LIN {X 0,Y 404.141,Z 498.144,A -85,B 0,C 180,E1 -10778.58,E2 -10778.58} C_VEL
LIN {X 0,Y 404.211,Z 498.134,A -85,B 0,C 180,E1 -10781.762,E2 -10781.762} C_VEL
LIN {X 0,Y 404.208,Z 498.138,A -85,B 0,C 180,E1 -10784.882,E2 -10784.882} C_VEL
LIN {X 0,Y 404.259,Z 498.127,A -85,B 0,C 180,E1 -10787.958,E2 -10787.958} C_VEL
LIN {X 0,Y 404.268,Z 498.129,A -85,B 0,C 180,E1 -10790.998,E2 -10790.998} C_VEL
LIN {X 0,Y 404.394,Z 498.111,A -85,B 0,C 180,E1 -10794.014,E2 -10794.014} C_VEL
LIN {X 0,Y 404.48,Z 498.1,A -85,B 0,C 180,E1 -10798.008,E2 -10798.008} C_VEL
LIN {X 0,Y 404.607,Z 498.084,A -85,B 0,C 180,E1 -10800,E2 -10800} C_VEL
LIN {X 0,Y 404.404,Z 498.112,A -85,B 0,C 180,E1 -10802.988,E2 -10802.988} C_VEL
LIN {X 0,Y 404.384,Z 498.112,A -85,B 0,C 180,E1 -10805.985,E2 -10805.985} C_VEL
LIN {X 0,Y 404.292,Z 498.126,A -85,B 0,C 180,E1 -10809.001,E2 -10809.001} C_VEL
LIN {X 0,Y 404.271,Z 498.126,A -85,B 0,C 180,E1 -10812.041,E2 -10812.041} C_VEL
LIN {X 0,Y 404.209,Z 498.136,A -85,B 0,C 180,E1 -10815.118,E2 -10815.118} C_VEL
LIN {X 0,Y 404.206,Z 498.135,A -85,B 0,C 180,E1 -10818.238,E2 -10818.238} C_VEL
LIN {X 0,Y 404.14,Z 498.144,A -85,B 0,C 180,E1 -10821.419,E2 -10821.419} C_VEL
LIN {X 0,Y 404.168,Z 498.142,A -85,B 0,C 180,E1 -10824.666,E2 -10824.666} C_VEL
LIN {X 0,Y 404.131,Z 498.144,A -85,B 0,C 180,E1 -10828.004,E2 -10828.004} C_VEL
LIN {X 0,Y 404.145,Z 498.143,A -85,B 0,C 180,E1 -10830.285,E2 -10830.285} C_VEL
LIN {X 0,Y 404.145,Z 498.142,A -85,B 0,C 180,E1 -10833.812,E2 -10833.812} C_VEL
LIN {X 0,Y 404.136,Z 498.147,A -85,B 0,C 180,E1 -10836.875,E2 -10836.875} C_VEL
LIN {X 0,Y 404.148,Z 498.145,A -85,B 0,C 180,E1 -10840.08,E2 -10840.08} C_VEL
LIN {X 0,Y 404.154,Z 498.142,A -85,B 0,C 180,E1 -10843.084,E2 -10843.084} C_VEL
LIN {X 0,Y 404.134,Z 498.16,A -85,B 0,C 180,E1 -10846.209,E2 -10846.209} C_VEL
LIN {X 0,Y 406.097,Z 507.927,A -85,B 0,C 180,E1 -10849.594,E2 -10849.594} C_VEL
LIN {X 0,Y 407.787,Z 516.569,A -85,B 0,C 180,E1 -10852.447,E2 -10852.447} C_VEL
LIN {X 0,Y 407.828,Z 520.057,A -85,B 0,C 180,E1 -10853.521,E2 -10853.521} C_VEL
LIN {X 0,Y 406.921,Z 529.958,A -85,B 0,C 180,E1 -10856.449,E2 -10856.449} C_VEL
LIN {X 0,Y 406.204,Z 539.849,A -85,B 0,C 180,E1 -10859.31,E2 -10859.31} C_VEL
LIN {X 0,Y 405.219,Z 553.615,A -85,B 0,C 180,E1 -10863.196,E2 -10863.196} C_VEL
LIN {X 0,Y 404.615,Z 565.406,A -85,B 0,C 180,E1 -10866.453,E2 -10866.453} C_VEL
LIN {X 0,Y 404,Z 579.554,A -85,B 0,C 180,E1 -10870.312,E2 -10870.312} C_VEL
LIN {X 0,Y 403.764,Z 586.685,A -85,B 0,C 180,E1 -10872.233,E2 -10872.233} C_VEL
LIN {X 0,Y 405.264,Z 601.573,A -85,B 0,C 180,E1 -10872.747,E2 -10872.747} C_VEL
LIN {X 0,Y 406.227,Z 614.758,A -85,B 0,C 180,E1 -10873.399,E2 -10873.399} C_VEL
LIN {X 0,Y 406.842,Z 625.399,A -85,B 0,C 180,E1 -10874.084,E2 -10874.084} C_VEL
LIN {X 0,Y 406.078,Z 636.59,A -85,B 0,C 180,E1 -10874.953,E2 -10874.953} C_VEL
LIN {X 0,Y 405.348,Z 646.907,A -85,B 0,C 180,E1 -10875.952,E2 -10875.952} C_VEL
LIN {X 0,Y 404.778,Z 654.204,A -85,B 0,C 180,E1 -10876.795,E2 -10876.795} C_VEL
LIN {X 0,Y 404.342,Z 660.999,A -85,B 0,C 180,E1 -10877.706,E2 -10877.706} C_VEL
LIN {X 0,Y 403.912,Z 668.935,A -85,B 0,C 180,E1 -10878.966,E2 -10878.966} C_VEL
LIN {X 0,Y 403.564,Z 676.692,A -85,B 0,C 180,E1 -10880.477,E2 -10880.477} C_VEL
LIN {X 0,Y 403.396,Z 682.935,A -85,B 0,C 180,E1 -10881.988,E2 -10881.988} C_VEL
LIN {X 0,Y 403.358,Z 687.287,A -85,B 0,C 180,E1 -10883.292,E2 -10883.292} C_VEL
LIN {X 0,Y 403.51,Z 691.675,A -85,B 0,C 180,E1 -10885.004,E2 -10885.004} C_VEL
LIN {X 0,Y 403.575,Z 693.612,A -85,B 0,C 180,E1 -10886.006,E2 -10886.006} C_VEL
LIN {X 0,Y 403.543,Z 695.082,A -85,B 0,C 180,E1 -10887.005,E2 -10887.005} C_VEL
LIN {X 0,Y 403.577,Z 696.088,A -85,B 0,C 180,E1 -10888.004,E2 -10888.004} C_VEL
LIN {X 0,Y 403.818,Z 696.903,A -85,B 0,C 180,E1 -10890,E2 -10890} C_VEL
LIN {X 0,Y 403.62,Z 696.63,A -85,B 0,C 180,E1 -10890.998,E2 -10890.998} C_VEL
LIN {X 0,Y 403.595,Z 695.93,A -85,B 0,C 180,E1 -10891.996,E2 -10891.996} C_VEL
LIN {X 0,Y 403.565,Z 694.822,A -85,B 0,C 180,E1 -10892.995,E2 -10892.995} C_VEL
LIN {X 0,Y 403.576,Z 692.346,A -85,B 0,C 180,E1 -10894.495,E2 -10894.495} C_VEL
LIN {X 0,Y 403.425,Z 688.813,A -85,B 0,C 180,E1 -10896,E2 -10896} C_VEL
LIN {X 0,Y 403.407,Z 684.179,A -85,B 0,C 180,E1 -10897.508,E2 -10897.508} C_VEL
LIN {X 0,Y 403.496,Z 678.319,A -85,B 0,C 180,E1 -10899.019,E2 -10899.019} C_VEL
LIN {X 0,Y 403.739,Z 671.062,A -85,B 0,C 180,E1 -10900.532,E2 -10900.532} C_VEL
LIN {X 0,Y 404.148,Z 663.731,A -85,B 0,C 180,E1 -10901.79,E2 -10901.79} C_VEL
LIN {X 0,Y 404.728,Z 654.992,A -85,B 0,C 180,E1 -10903.047,E2 -10903.047} C_VEL
LIN {X 0,Y 405.372,Z 645.507,A -85,B 0,C 180,E1 -10904.175,E2 -10904.175} C_VEL
LIN {X 0,Y 406.273,Z 633.869,A -85,B 0,C 180,E1 -10905.296,E2 -10905.296} C_VEL
LIN {X 0,Y 406.924,Z 624.366,A -85,B 0,C 180,E1 -10906.042,E2 -10906.042} C_VEL
LIN {X 0,Y 406.386,Z 614.636,A -85,B 0,C 180,E1 -10906.709,E2 -10906.709} C_VEL
LIN {X 0,Y 405.749,Z 600.808,A -85,B 0,C 180,E1 -10907.444,E2 -10907.444} C_VEL
LIN {X 0,Y 404.415,Z 587.584,A -85,B 0,C 180,E1 -10907.975,E2 -10907.975} C_VEL
LIN {X 0,Y 403.758,Z 582.357,A -85,B 0,C 180,E1 -10908.164,E2 -10908.164} C_VEL
LIN {X 0,Y 404.09,Z 568.944,A -85,B 0,C 180,E1 -10911.69,E2 -10911.69} C_VEL
LIN {X 0,Y 404.645,Z 555.051,A -85,B 0,C 180,E1 -10915.424,E2 -10915.424} C_VEL
LIN {X 0,Y 405.304,Z 541.989,A -85,B 0,C 180,E1 -10919.047,E2 -10919.047} C_VEL
LIN {X 0,Y 406.089,Z 530.165,A -85,B 0,C 180,E1 -10922.446,E2 -10922.446} C_VEL
LIN {X 0,Y 407.046,Z 518.566,A -85,B 0,C 180,E1 -10925.948,E2 -10925.948} C_VEL
LIN {X 0,Y 407.158,Z 513.919,A -85,B 0,C 180,E1 -10927.438,E2 -10927.438} C_VEL
LIN {X 0,Y 405.718,Z 505.699,A -85,B 0,C 180,E1 -10930.343,E2 -10930.343} C_VEL
LIN {X 0,Y 404.151,Z 498.147,A -85,B 0,C 180,E1 -10933.287,E2 -10933.287} C_VEL
LIN {X 0,Y 404.156,Z 498.146,A -85,B 0,C 180,E1 -10936.916,E2 -10936.916} C_VEL
LIN {X 0,Y 404.171,Z 498.141,A -85,B 0,C 180,E1 -10939.956,E2 -10939.956} C_VEL
LIN {X 0,Y 404.138,Z 498.145,A -85,B 0,C 180,E1 -10943.125,E2 -10943.125} C_VEL
LIN {X 0,Y 404.147,Z 498.142,A -85,B 0,C 180,E1 -10946.188,E2 -10946.188} C_VEL
LIN {X 0,Y 404.148,Z 498.144,A -85,B 0,C 180,E1 -10949.715,E2 -10949.715} C_VEL
LIN {X 0,Y 404.198,Z 498.133,A -85,B 0,C 180,E1 -10953.123,E2 -10953.123} C_VEL
LIN {X 0,Y 404.18,Z 498.137,A -85,B 0,C 180,E1 -10955.335,E2 -10955.335} C_VEL
LIN {X 0,Y 404.142,Z 498.14,A -85,B 0,C 180,E1 -10958.581,E2 -10958.581} C_VEL
LIN {X 0,Y 404.212,Z 498.132,A -85,B 0,C 180,E1 -10961.762,E2 -10961.762} C_VEL
LIN {X 0,Y 404.21,Z 498.132,A -85,B 0,C 180,E1 -10964.882,E2 -10964.882} C_VEL
LIN {X 0,Y 404.26,Z 498.128,A -85,B 0,C 180,E1 -10967.959,E2 -10967.959} C_VEL
LIN {X 0,Y 404.437,Z 498.103,A -85,B 0,C 180,E1 -10972.1,E2 -10972.1} C_VEL
LIN {X 0,Y 404.428,Z 498.108,A -85,B 0,C 180,E1 -10974.015,E2 -10974.015} C_VEL
LIN {X 0,Y 404.482,Z 498.101,A -85,B 0,C 180,E1 -10978.009,E2 -10978.009} C_VEL
LIN {X 0,Y 404.612,Z 498.086,A -85,B 0,C 180,E1 -10980,E2 -10980} C_VEL
LIN {X 0,Y 404.419,Z 498.111,A -85,B 0,C 180,E1 -10982.989,E2 -10982.989} C_VEL
LIN {X 0,Y 404.35,Z 498.114,A -85,B 0,C 180,E1 -10986.534,E2 -10986.534} C_VEL
LIN {X 0,Y 404.293,Z 498.123,A -85,B 0,C 180,E1 -10989.001,E2 -10989.001} C_VEL
LIN {X 0,Y 404.261,Z 498.131,A -85,B 0,C 180,E1 -10992.042,E2 -10992.042} C_VEL
LIN {X 0,Y 404.213,Z 498.136,A -85,B 0,C 180,E1 -10995.118,E2 -10995.118} C_VEL
LIN {X 0,Y 404.259,Z 498.134,A -85,B 0,C 180,E1 -10996.745,E2 -10996.745} C_VEL
LIN {X 0,Y 408.406,Z 510.86,A -85,B 0,C 180,E1 -10997.786,E2 -10997.786} C_VEL
LIN {X 0,Y 409.398,Z 514.616,A -85,B 0,C 180,E1 -10998.129,E2 -10998.129} C_VEL
LIN {X 0,Y 408.929,Z 525.453,A -85,B 0,C 180,E1 -10999.059,E2 -10999.059} C_VEL
LIN {X 0,Y 408.19,Z 535.615,A -85,B 0,C 180,E1 -11000.142,E2 -11000.142} C_VEL
LIN {X 0,Y 407.382,Z 545.671,A -85,B 0,C 180,E1 -11001.479,E2 -11001.479} C_VEL
LIN {X 0,Y 406.617,Z 554.21,A -85,B 0,C 180,E1 -11002.886,E2 -11002.886} C_VEL
LIN {X 0,Y 406.019,Z 560.977,A -85,B 0,C 180,E1 -11004.274,E2 -11004.274} C_VEL
LIN {X 0,Y 405.502,Z 566.524,A -85,B 0,C 180,E1 -11005.677,E2 -11005.677} C_VEL
LIN {X 0,Y 405.001,Z 571.46,A -85,B 0,C 180,E1 -11007.261,E2 -11007.261} C_VEL
LIN {X 0,Y 404.571,Z 575.675,A -85,B 0,C 180,E1 -11009.105,E2 -11009.105} C_VEL
LIN {X 0,Y 404.343,Z 577.544,A -85,B 0,C 180,E1 -11010.269,E2 -11010.269} C_VEL
LIN {X 0,Y 404.164,Z 578.987,A -85,B 0,C 180,E1 -11011.563,E2 -11011.563} C_VEL
LIN {X 0,Y 404.021,Z 579.832,A -85,B 0,C 180,E1 -11013.387,E2 -11013.387} C_VEL
LIN {X 0,Y 403.999,Z 579.409,A -85,B 0,C 180,E1 -11015.153,E2 -11015.153} C_VEL
LIN {X 0,Y 404.036,Z 577.843,A -85,B 0,C 180,E1 -11016.855,E2 -11016.855} C_VEL
LIN {X 0,Y 404.242,Z 574.712,A -85,B 0,C 180,E1 -11018.748,E2 -11018.748} C_VEL
LIN {X 0,Y 404.633,Z 569.886,A -85,B 0,C 180,E1 -11020.661,E2 -11020.661} C_VEL
LIN {X 0,Y 404.958,Z 565.075,A -85,B 0,C 180,E1 -11022.102,E2 -11022.102} C_VEL
LIN {X 0,Y 405.363,Z 559.33,A -85,B 0,C 180,E1 -11023.489,E2 -11023.489} C_VEL
LIN {X 0,Y 405.978,Z 551.93,A -85,B 0,C 180,E1 -11024.94,E2 -11024.94} C_VEL
LIN {X 0,Y 406.592,Z 543.052,A -85,B 0,C 180,E1 -11026.347,E2 -11026.347} C_VEL
LIN {X 0,Y 407.271,Z 533.218,A -85,B 0,C 180,E1 -11027.609,E2 -11027.609} C_VEL
LIN {X 0,Y 407.904,Z 522.41,A -85,B 0,C 180,E1 -11028.733,E2 -11028.733} C_VEL
LIN {X 0,Y 408.384,Z 513.674,A -85,B 0,C 180,E1 -11029.47,E2 -11029.47} C_VEL
LIN {X 0,Y 405.738,Z 503.665,A -85,B 0,C 180,E1 -11030.302,E2 -11030.302} C_VEL
LIN {X 0,Y 404.159,Z 498.143,A -85,B 0,C 180,E1 -11030.722,E2 -11030.722} C_VEL
LIN {X 0,Y 404.146,Z 498.145,A -85,B 0,C 180,E1 -11033.754,E2 -11033.754} C_VEL
LIN {X 0,Y 404.176,Z 498.137,A -85,B 0,C 180,E1 -11036.58,E2 -11036.58} C_VEL
LIN {X 0,Y 404.168,Z 498.138,A -85,B 0,C 180,E1 -11040.395,E2 -11040.395} C_VEL
LIN {X 0,Y 404.199,Z 498.138,A -85,B 0,C 180,E1 -11043.123,E2 -11043.123} C_VEL
LIN {X 0,Y 404.175,Z 498.141,A -85,B 0,C 180,E1 -11045.334,E2 -11045.334} C_VEL
LIN {X 0,Y 404.144,Z 498.142,A -85,B 0,C 180,E1 -11048.581,E2 -11048.581} C_VEL
LIN {X 0,Y 404.21,Z 498.136,A -85,B 0,C 180,E1 -11051.762,E2 -11051.762} C_VEL
LIN {X 0,Y 404.211,Z 498.135,A -85,B 0,C 180,E1 -11054.882,E2 -11054.882} C_VEL
LIN {X 0,Y 404.262,Z 498.128,A -85,B 0,C 180,E1 -11057.958,E2 -11057.958} C_VEL
LIN {X 0,Y 404.272,Z 498.129,A -85,B 0,C 180,E1 -11060.998,E2 -11060.998} C_VEL
LIN {X 0,Y 404.387,Z 498.112,A -85,B 0,C 180,E1 -11064.014,E2 -11064.014} C_VEL
LIN {X 0,Y 404.485,Z 498.1,A -85,B 0,C 180,E1 -11068.008,E2 -11068.008} C_VEL
LIN {X 0,Y 404.606,Z 498.085,A -85,B 0,C 180,E1 -11070,E2 -11070} C_VEL
LIN {X 0,Y 404.413,Z 498.111,A -85,B 0,C 180,E1 -11072.988,E2 -11072.988} C_VEL
LIN {X 0,Y 404.386,Z 498.112,A -85,B 0,C 180,E1 -11075.985,E2 -11075.985} C_VEL
LIN {X 0,Y 404.271,Z 498.129,A -85,B 0,C 180,E1 -11079.001,E2 -11079.001} C_VEL
LIN {X 0,Y 404.261,Z 498.127,A -85,B 0,C 180,E1 -11082.041,E2 -11082.041} C_VEL
LIN {X 0,Y 404.205,Z 498.136,A -85,B 0,C 180,E1 -11085.267,E2 -11085.267} C_VEL
LIN {X 0,Y 403.533,Z 498.219,A -85,B 0,C 180,E1 -11086.098,E2 -11086.098} C_VEL
LIN {X 0,Y 400.696,Z 498.575,A -85,B 0,C 180,E1 -11087.449,E2 -11087.449} C_VEL
LIN {X 0,Y 398.29,Z 498.876,A -85,B 0,C 180,E1 -11088.54,E2 -11088.54} C_VEL
LIN {X 0,Y 397.243,Z 499.004,A -85,B 0,C 180,E1 -11089.384,E2 -11089.384} C_VEL
LIN {X 0,Y 397.15,Z 499.014,A -85,B 0,C 180,E1 -11089.67,E2 -11089.67} C_VEL
LIN {X 0,Y 397.139,Z 499.017,A -85,B 0,C 180,E1 -11093.04,E2 -11093.04} C_VEL
LIN {X 0,Y 397.107,Z 499.017,A -85,B 0,C 180,E1 -11096.26,E2 -11096.26} C_VEL
LIN {X 0,Y 397.123,Z 499.018,A -85,B 0,C 180,E1 -11099.704,E2 -11099.704} C_VEL
LIN {X 0,Y 397.118,Z 499.02,A -85,B 0,C 180,E1 -11103.273,E2 -11103.273} C_VEL
LIN {X 0,Y 397.111,Z 499.019,A -85,B 0,C 180,E1 -11105.734,E2 -11105.734} C_VEL
LIN {X 0,Y 397.098,Z 499.022,A -85,B 0,C 180,E1 -11108.855,E2 -11108.855} C_VEL
LIN {X 0,Y 397.06,Z 499.024,A -85,B 0,C 180,E1 -11112.268,E2 -11112.268} C_VEL
LIN {X 0,Y 397.09,Z 499.024,A -85,B 0,C 180,E1 -11115.069,E2 -11115.069} C_VEL
LIN {X 0,Y 397.065,Z 499.023,A -85,B 0,C 180,E1 -11118.022,E2 -11118.022} C_VEL
LIN {X 0,Y 397.127,Z 499.019,A -85,B 0,C 180,E1 -11121.139,E2 -11121.139} C_VEL
LIN {X 0,Y 397.122,Z 499.018,A -85,B 0,C 180,E1 -11124.496,E2 -11124.496} C_VEL
LIN {X 0,Y 397.081,Z 499.022,A -85,B 0,C 180,E1 -11127.928,E2 -11127.928} C_VEL
LIN {X 0,Y 397.125,Z 499.017,A -85,B 0,C 180,E1 -11131.456,E2 -11131.456} C_VEL
LIN {X 0,Y 397.154,Z 499.014,A -85,B 0,C 180,E1 -11134.488,E2 -11134.488} C_VEL
LIN {X 0,Y 397.099,Z 499.018,A -85,B 0,C 180,E1 -11138.181,E2 -11138.181} C_VEL
LIN {X 0,Y 397.164,Z 499.013,A -85,B 0,C 180,E1 -11141.426,E2 -11141.426} C_VEL
LIN {X 0,Y 397.181,Z 499.011,A -85,B 0,C 180,E1 -11144.608,E2 -11144.608} C_VEL
LIN {X 0,Y 397.222,Z 499.004,A -85,B 0,C 180,E1 -11147.742,E2 -11147.742} C_VEL
LIN {X 0,Y 397.238,Z 499.006,A -85,B 0,C 180,E1 -11150.837,E2 -11150.837} C_VEL
LIN {X 0,Y 397.346,Z 498.988,A -85,B 0,C 180,E1 -11153.908,E2 -11153.908} C_VEL
LIN {X 0,Y 397.449,Z 498.976,A -85,B 0,C 180,E1 -11157.973,E2 -11157.973} C_VEL
LIN {X 0,Y 397.577,Z 498.96,A -85,B 0,C 180,E1 -11160,E2 -11160} C_VEL
LIN {X 0,Y 397.337,Z 498.992,A -85,B 0,C 180,E1 -11163.041,E2 -11163.041} C_VEL
LIN {X 0,Y 397.335,Z 498.99,A -85,B 0,C 180,E1 -11166.092,E2 -11166.092} C_VEL
LIN {X 0,Y 397.254,Z 499.002,A -85,B 0,C 180,E1 -11169.162,E2 -11169.162} C_VEL
LIN {X 0,Y 397.23,Z 499.004,A -85,B 0,C 180,E1 -11172.258,E2 -11172.258} C_VEL
LIN {X 0,Y 397.181,Z 499.011,A -85,B 0,C 180,E1 -11175.392,E2 -11175.392} C_VEL
LIN {X 0,Y 397.16,Z 499.014,A -85,B 0,C 180,E1 -11178.573,E2 -11178.573} C_VEL
LIN {X 0,Y 397.098,Z 499.019,A -85,B 0,C 180,E1 -11181.818,E2 -11181.818} C_VEL
LIN {X 0,Y 397.125,Z 499.018,A -85,B 0,C 180,E1 -11185.134,E2 -11185.134} C_VEL
LIN {X 0,Y 397.079,Z 499.025,A -85,B 0,C 180,E1 -11188.547,E2 -11188.547} C_VEL
LIN {X 0,Y 397.082,Z 499.02,A -85,B 0,C 180,E1 -11191.836,E2 -11191.836} C_VEL
LIN {X 0,Y 397.126,Z 499.019,A -85,B 0,C 180,E1 -11194.493,E2 -11194.493} C_VEL
LIN {X 0,Y 397.099,Z 499.02,A -85,B 0,C 180,E1 -11198.275,E2 -11198.275} C_VEL
LIN {X 0,Y 397.09,Z 499.024,A -85,B 0,C 180,E1 -11200.909,E2 -11200.909} C_VEL
LIN {X 0,Y 397.102,Z 499.019,A -85,B 0,C 180,E1 -11203.648,E2 -11203.648} C_VEL
LIN {X 0,Y 397.122,Z 499.123,A -85,B 0,C 180,E1 -11205.91,E2 -11205.91} C_VEL
LIN {X 0,Y 399.047,Z 508.804,A -85,B 0,C 180,E1 -11209.334,E2 -11209.334} C_VEL
LIN {X 0,Y 400.847,Z 518.125,A -85,B 0,C 180,E1 -11212.463,E2 -11212.463} C_VEL
LIN {X 0,Y 400.738,Z 522.352,A -85,B 0,C 180,E1 -11213.778,E2 -11213.778} C_VEL
LIN {X 0,Y 399.751,Z 532.996,A -85,B 0,C 180,E1 -11216.975,E2 -11216.975} C_VEL
LIN {X 0,Y 398.957,Z 543.459,A -85,B 0,C 180,E1 -11220.044,E2 -11220.044} C_VEL
LIN {X 0,Y 398.034,Z 556.584,A -85,B 0,C 180,E1 -11223.806,E2 -11223.806} C_VEL
LIN {X 0,Y 397.407,Z 568.298,A -85,B 0,C 180,E1 -11227.104,E2 -11227.104} C_VEL
LIN {X 0,Y 396.82,Z 581.904,A -85,B 0,C 180,E1 -11230.874,E2 -11230.874} C_VEL
LIN {X 0,Y 396.676,Z 585.78,A -85,B 0,C 180,E1 -11231.938,E2 -11231.938} C_VEL
LIN {X 0,Y 398.191,Z 600.26,A -85,B 0,C 180,E1 -11232.449,E2 -11232.449} C_VEL
LIN {X 0,Y 399.15,Z 613.084,A -85,B 0,C 180,E1 -11233.087,E2 -11233.087} C_VEL
LIN {X 0,Y 399.754,Z 623.972,A -85,B 0,C 180,E1 -11233.794,E2 -11233.794} C_VEL
LIN {X 0,Y 399.239,Z 633.846,A -85,B 0,C 180,E1 -11234.559,E2 -11234.559} C_VEL
LIN {X 0,Y 398.35,Z 645.631,A -85,B 0,C 180,E1 -11235.7,E2 -11235.7} C_VEL
LIN {X 0,Y 397.71,Z 654.208,A -85,B 0,C 180,E1 -11236.719,E2 -11236.719} C_VEL
LIN {X 0,Y 397.111,Z 663.135,A -85,B 0,C 180,E1 -11237.998,E2 -11237.998} C_VEL
LIN {X 0,Y 396.72,Z 670.534,A -85,B 0,C 180,E1 -11239.28,E2 -11239.28} C_VEL
LIN {X 0,Y 396.406,Z 677.823,A -85,B 0,C 180,E1 -11240.819,E2 -11240.819} C_VEL
LIN {X 0,Y 396.309,Z 683.639,A -85,B 0,C 180,E1 -11242.357,E2 -11242.357} C_VEL
LIN {X 0,Y 396.331,Z 688.204,A -85,B 0,C 180,E1 -11243.893,E2 -11243.893} C_VEL
LIN {X 0,Y 396.464,Z 690.607,A -85,B 0,C 180,E1 -11244.915,E2 -11244.915} C_VEL
LIN {X 0,Y 396.539,Z 692.553,A -85,B 0,C 180,E1 -11245.935,E2 -11245.935} C_VEL
LIN {X 0,Y 396.506,Z 694.036,A -85,B 0,C 180,E1 -11246.952,E2 -11246.952} C_VEL
LIN {X 0,Y 396.542,Z 695.051,A -85,B 0,C 180,E1 -11247.969,E2 -11247.969} C_VEL
LIN {X 0,Y 396.795,Z 695.873,A -85,B 0,C 180,E1 -11250,E2 -11250} C_VEL
LIN {X 0,Y 396.589,Z 695.609,A -85,B 0,C 180,E1 -11251.016,E2 -11251.016} C_VEL
LIN {X 0,Y 396.556,Z 694.912,A -85,B 0,C 180,E1 -11252.031,E2 -11252.031} C_VEL
LIN {X 0,Y 396.572,Z 692.289,A -85,B 0,C 180,E1 -11254.065,E2 -11254.065} C_VEL
LIN {X 0,Y 396.373,Z 689.098,A -85,B 0,C 180,E1 -11255.596,E2 -11255.596} C_VEL
LIN {X 0,Y 396.34,Z 684.847,A -85,B 0,C 180,E1 -11257.13,E2 -11257.13} C_VEL
LIN {X 0,Y 396.411,Z 678.397,A -85,B 0,C 180,E1 -11258.924,E2 -11258.924} C_VEL
LIN {X 0,Y 396.625,Z 671.39,A -85,B 0,C 180,E1 -11260.465,E2 -11260.465} C_VEL
LIN {X 0,Y 397.113,Z 662.782,A -85,B 0,C 180,E1 -11262.002,E2 -11262.002} C_VEL
LIN {X 0,Y 397.662,Z 654.059,A -85,B 0,C 180,E1 -11263.283,E2 -11263.283} C_VEL
LIN {X 0,Y 398.556,Z 643.445,A -85,B 0,C 180,E1 -11264.553,E2 -11264.553} C_VEL
LIN {X 0,Y 399.413,Z 633.058,A -85,B 0,C 180,E1 -11265.565,E2 -11265.565} C_VEL
LIN {X 0,Y 399.956,Z 625.373,A -85,B 0,C 180,E1 -11266.198,E2 -11266.198} C_VEL
LIN {X 0,Y 399.455,Z 614.004,A -85,B 0,C 180,E1 -11267.008,E2 -11267.008} C_VEL
LIN {X 0,Y 398.847,Z 600.684,A -85,B 0,C 180,E1 -11267.747,E2 -11267.747} C_VEL
LIN {X 0,Y 397.502,Z 586.889,A -85,B 0,C 180,E1 -11268.332,E2 -11268.332} C_VEL
LIN {X 0,Y 396.685,Z 581.208,A -85,B 0,C 180,E1 -11268.53,E2 -11268.53} C_VEL
LIN {X 0,Y 397.056,Z 567.967,A -85,B 0,C 180,E1 -11272.095,E2 -11272.095} C_VEL
LIN {X 0,Y 397.642,Z 555.002,A -85,B 0,C 180,E1 -11275.659,E2 -11275.659} C_VEL
LIN {X 0,Y 398.254,Z 543.102,A -85,B 0,C 180,E1 -11279.032,E2 -11279.032} C_VEL
LIN {X 0,Y 399.132,Z 530.894,A -85,B 0,C 180,E1 -11282.624,E2 -11282.624} C_VEL
LIN {X 0,Y 400.103,Z 519.649,A -85,B 0,C 180,E1 -11286.098,E2 -11286.098} C_VEL
LIN {X 0,Y 400.33,Z 516.239,A -85,B 0,C 180,E1 -11287.199,E2 -11287.199} C_VEL
LIN {X 0,Y 399.018,Z 508.383,A -85,B 0,C 180,E1 -11290.008,E2 -11290.008} C_VEL
LIN {X 0,Y 397.547,Z 501.176,A -85,B 0,C 180,E1 -11292.829,E2 -11292.829} C_VEL
LIN {X 0,Y 397.106,Z 499.027,A -85,B 0,C 180,E1 -11293.736,E2 -11293.736} C_VEL
LIN {X 0,Y 397.105,Z 499.026,A -85,B 0,C 180,E1 -11296.521,E2 -11296.521} C_VEL
LIN {X 0,Y 397.116,Z 499.021,A -85,B 0,C 180,E1 -11300.423,E2 -11300.423} C_VEL
LIN {X 0,Y 397.11,Z 499.02,A -85,B 0,C 180,E1 -11304.266,E2 -11304.266} C_VEL
LIN {X 0,Y 397.117,Z 499.019,A -85,B 0,C 180,E1 -11306.727,E2 -11306.727} C_VEL
LIN {X 0,Y 397.127,Z 499.014,A -85,B 0,C 180,E1 -11310.296,E2 -11310.296} C_VEL
LIN {X 0,Y 397.197,Z 499.006,A -85,B 0,C 180,E1 -11312.61,E2 -11312.61} C_VEL
LIN {X 0,Y 397.135,Z 499.012,A -85,B 0,C 180,E1 -11315.982,E2 -11315.982} C_VEL
LIN {X 0,Y 397.142,Z 499.013,A -85,B 0,C 180,E1 -11319.705,E2 -11319.705} C_VEL
LIN {X 0,Y 397.185,Z 499.01,A -85,B 0,C 180,E1 -11322.845,E2 -11322.845} C_VEL
LIN {X 0,Y 397.232,Z 499.005,A -85,B 0,C 180,E1 -11326.703,E2 -11326.703} C_VEL
LIN {X 0,Y 397.221,Z 499.007,A -85,B 0,C 180,E1 -11329.809,E2 -11329.809} C_VEL
LIN {X 0,Y 397.369,Z 498.987,A -85,B 0,C 180,E1 -11332.889,E2 -11332.889} C_VEL
LIN {X 0,Y 397.253,Z 498.998,A -85,B 0,C 180,E1 -11334.925,E2 -11334.925} C_VEL
LIN {X 0,Y 397.45,Z 498.976,A -85,B 0,C 180,E1 -11337.974,E2 -11337.974} C_VEL
LIN {X 0,Y 397.581,Z 498.961,A -85,B 0,C 180,E1 -11340,E2 -11340} C_VEL
LIN {X 0,Y 397.378,Z 498.988,A -85,B 0,C 180,E1 -11343.042,E2 -11343.042} C_VEL
LIN {X 0,Y 397.306,Z 498.991,A -85,B 0,C 180,E1 -11346.527,E2 -11346.527} C_VEL
LIN {X 0,Y 397.256,Z 499,A -85,B 0,C 180,E1 -11349.162,E2 -11349.162} C_VEL
LIN {X 0,Y 397.224,Z 499.009,A -85,B 0,C 180,E1 -11352.258,E2 -11352.258} C_VEL
LIN {X 0,Y 397.191,Z 499.013,A -85,B 0,C 180,E1 -11355.918,E2 -11355.918} C_VEL
LIN {X 0,Y 397.217,Z 499.129,A -85,B 0,C 180,E1 -11356.379,E2 -11356.379} C_VEL
LIN {X 0,Y 401.529,Z 512.126,A -85,B 0,C 180,E1 -11357.469,E2 -11357.469} C_VEL
LIN {X 0,Y 402.748,Z 516.55,A -85,B 0,C 180,E1 -11357.887,E2 -11357.887} C_VEL
LIN {X 0,Y 402.127,Z 527.968,A -85,B 0,C 180,E1 -11358.907,E2 -11358.907} C_VEL
LIN {X 0,Y 401.341,Z 538.575,A -85,B 0,C 180,E1 -11360.1,E2 -11360.1} C_VEL
LIN {X 0,Y 400.526,Z 547.771,A -85,B 0,C 180,E1 -11361.378,E2 -11361.378} C_VEL
LIN {X 0,Y 399.735,Z 555.793,A -85,B 0,C 180,E1 -11362.756,E2 -11362.756} C_VEL
LIN {X 0,Y 398.97,Z 563.649,A -85,B 0,C 180,E1 -11364.454,E2 -11364.454} C_VEL
LIN {X 0,Y 398.343,Z 569.823,A -85,B 0,C 180,E1 -11366.173,E2 -11366.173} C_VEL
LIN {X 0,Y 397.843,Z 574.613,A -85,B 0,C 180,E1 -11367.961,E2 -11367.961} C_VEL
LIN {X 0,Y 397.436,Z 577.893,A -85,B 0,C 180,E1 -11369.679,E2 -11369.679} C_VEL
LIN {X 0,Y 397.259,Z 579.438,A -85,B 0,C 180,E1 -11370.867,E2 -11370.867} C_VEL
LIN {X 0,Y 397.087,Z 580.431,A -85,B 0,C 180,E1 -11372.071,E2 -11372.071} C_VEL
LIN {X 0,Y 397.006,Z 580.885,A -85,B 0,C 180,E1 -11373.693,E2 -11373.693} C_VEL
LIN {X 0,Y 397.002,Z 580.025,A -85,B 0,C 180,E1 -11375.746,E2 -11375.746} C_VEL
LIN {X 0,Y 397.043,Z 578.454,A -85,B 0,C 180,E1 -11377.199,E2 -11377.199} C_VEL
LIN {X 0,Y 397.238,Z 575.543,A -85,B 0,C 180,E1 -11378.88,E2 -11378.88} C_VEL
LIN {X 0,Y 397.663,Z 570.612,A -85,B 0,C 180,E1 -11380.838,E2 -11380.838} C_VEL
LIN {X 0,Y 398.085,Z 565.076,A -85,B 0,C 180,E1 -11382.477,E2 -11382.477} C_VEL
LIN {X 0,Y 398.64,Z 557.594,A -85,B 0,C 180,E1 -11384.195,E2 -11384.195} C_VEL
LIN {X 0,Y 399.292,Z 549.75,A -85,B 0,C 180,E1 -11385.635,E2 -11385.635} C_VEL
LIN {X 0,Y 399.971,Z 540.08,A -85,B 0,C 180,E1 -11387.072,E2 -11387.072} C_VEL
LIN {X 0,Y 400.688,Z 529.022,A -85,B 0,C 180,E1 -11388.385,E2 -11388.385} C_VEL
LIN {X 0,Y 401.335,Z 518.926,A -85,B 0,C 180,E1 -11389.348,E2 -11389.348} C_VEL
LIN {X 0,Y 401.318,Z 513.838,A -85,B 0,C 180,E1 -11389.776,E2 -11389.776} C_VEL
LIN {X 0,Y 398.034,Z 502.298,A -85,B 0,C 180,E1 -11390.734,E2 -11390.734} C_VEL
LIN {X 0,Y 397.112,Z 499.022,A -85,B 0,C 180,E1 -11390.978,E2 -11390.978} C_VEL
LIN {X 0,Y 397.124,Z 499.016,A -85,B 0,C 180,E1 -11394.497,E2 -11394.497} C_VEL
LIN {X 0,Y 397.084,Z 499.023,A -85,B 0,C 180,E1 -11397.929,E2 -11397.929} C_VEL
LIN {X 0,Y 397.127,Z 499.02,A -85,B 0,C 180,E1 -11401.456,E2 -11401.456} C_VEL
LIN {X 0,Y 397.156,Z 499.012,A -85,B 0,C 180,E1 -11404.488,E2 -11404.488} C_VEL
LIN {X 0,Y 397.101,Z 499.019,A -85,B 0,C 180,E1 -11408.181,E2 -11408.181} C_VEL
LIN {X 0,Y 397.163,Z 499.015,A -85,B 0,C 180,E1 -11411.426,E2 -11411.426} C_VEL
LIN {X 0,Y 397.184,Z 499.009,A -85,B 0,C 180,E1 -11414.608,E2 -11414.608} C_VEL
LIN {X 0,Y 397.225,Z 499.006,A -85,B 0,C 180,E1 -11417.742,E2 -11417.742} C_VEL
LIN {X 0,Y 397.241,Z 499.003,A -85,B 0,C 180,E1 -11420.838,E2 -11420.838} C_VEL
LIN {X 0,Y 397.338,Z 498.99,A -85,B 0,C 180,E1 -11423.908,E2 -11423.908} C_VEL
LIN {X 0,Y 397.454,Z 498.976,A -85,B 0,C 180,E1 -11427.973,E2 -11427.973} C_VEL
LIN {X 0,Y 397.576,Z 498.96,A -85,B 0,C 180,E1 -11430,E2 -11430} C_VEL
LIN {X 0,Y 397.372,Z 498.989,A -85,B 0,C 180,E1 -11433.041,E2 -11433.041} C_VEL
LIN {X 0,Y 397.337,Z 498.989,A -85,B 0,C 180,E1 -11436.092,E2 -11436.092} C_VEL
LIN {X 0,Y 397.241,Z 499.005,A -85,B 0,C 180,E1 -11439.162,E2 -11439.162} C_VEL
LIN {X 0,Y 397.224,Z 499.003,A -85,B 0,C 180,E1 -11442.258,E2 -11442.258} C_VEL
LIN {X 0,Y 397.184,Z 499.011,A -85,B 0,C 180,E1 -11445.392,E2 -11445.392} C_VEL
LIN {X 0,Y 397.162,Z 499.012,A -85,B 0,C 180,E1 -11448.573,E2 -11448.573} C_VEL
LIN {X 0,Y 397.15,Z 499.014,A -85,B 0,C 180,E1 -11449.67,E2 -11449.67} C_VEL
LIN {X 0,Y 396.457,Z 499.1,A -85,B 0,C 180,E1 -11450.515,E2 -11450.515} C_VEL
LIN {X 0,Y 393.582,Z 499.458,A -85,B 0,C 180,E1 -11451.89,E2 -11451.89} C_VEL
LIN {X 0,Y 391.166,Z 499.761,A -85,B 0,C 180,E1 -11453.001,E2 -11453.001} C_VEL
LIN {X 0,Y 390.138,Z 499.887,A -85,B 0,C 180,E1 -11453.86,E2 -11453.86} C_VEL
LIN {X 0,Y 390.059,Z 499.895,A -85,B 0,C 180,E1 -11454.151,E2 -11454.151} C_VEL
LIN {X 0,Y 390.078,Z 499.895,A -85,B 0,C 180,E1 -11456.771,E2 -11456.771} C_VEL
LIN {X 0,Y 390.041,Z 499.898,A -85,B 0,C 180,E1 -11460.3,E2 -11460.3} C_VEL
LIN {X 0,Y 390.072,Z 499.895,A -85,B 0,C 180,E1 -11464.024,E2 -11464.024} C_VEL
LIN {X 0,Y 390.043,Z 499.899,A -85,B 0,C 180,E1 -11467.55,E2 -11467.55} C_VEL
LIN {X 0,Y 390.021,Z 499.904,A -85,B 0,C 180,E1 -11470.814,E2 -11470.814} C_VEL
LIN {X 0,Y 390.055,Z 499.896,A -85,B 0,C 180,E1 -11473.885,E2 -11473.885} C_VEL
LIN {X 0,Y 390.059,Z 499.9,A -85,B 0,C 180,E1 -11476.789,E2 -11476.789} C_VEL
LIN {X 0,Y 390.059,Z 499.897,A -85,B 0,C 180,E1 -11479.56,E2 -11479.56} C_VEL
LIN {X 0,Y 390.044,Z 499.899,A -85,B 0,C 180,E1 -11482.449,E2 -11482.449} C_VEL
LIN {X 0,Y 390.071,Z 499.894,A -85,B 0,C 180,E1 -11485.975,E2 -11485.975} C_VEL
LIN {X 0,Y 390.05,Z 499.897,A -85,B 0,C 180,E1 -11489.869,E2 -11489.869} C_VEL
LIN {X 0,Y 390.115,Z 499.892,A -85,B 0,C 180,E1 -11493.231,E2 -11493.231} C_VEL
LIN {X 0,Y 390.07,Z 499.897,A -85,B 0,C 180,E1 -11496.763,E2 -11496.763} C_VEL
LIN {X 0,Y 390.106,Z 499.89,A -85,B 0,C 180,E1 -11499.983,E2 -11499.983} C_VEL
LIN {X 0,Y 390.141,Z 499.888,A -85,B 0,C 180,E1 -11503.248,E2 -11503.248} C_VEL
LIN {X 0,Y 390.197,Z 499.881,A -85,B 0,C 180,E1 -11506.561,E2 -11506.561} C_VEL
LIN {X 0,Y 390.17,Z 499.882,A -85,B 0,C 180,E1 -11509.623,E2 -11509.623} C_VEL
LIN {X 0,Y 390.269,Z 499.873,A -85,B 0,C 180,E1 -11512.758,E2 -11512.758} C_VEL
LIN {X 0,Y 390.219,Z 499.879,A -85,B 0,C 180,E1 -11514.833,E2 -11514.833} C_VEL
LIN {X 0,Y 390.418,Z 499.851,A -85,B 0,C 180,E1 -11517.936,E2 -11517.936} C_VEL
LIN {X 0,Y 390.546,Z 499.835,A -85,B 0,C 180,E1 -11520,E2 -11520} C_VEL
LIN {X 0,Y 390.274,Z 499.872,A -85,B 0,C 180,E1 -11523.097,E2 -11523.097} C_VEL
LIN {X 0,Y 390.288,Z 499.868,A -85,B 0,C 180,E1 -11526.202,E2 -11526.202} C_VEL
LIN {X 0,Y 390.207,Z 499.88,A -85,B 0,C 180,E1 -11529.329,E2 -11529.329} C_VEL
LIN {X 0,Y 390.179,Z 499.883,A -85,B 0,C 180,E1 -11532.483,E2 -11532.483} C_VEL
LIN {X 0,Y 390.141,Z 499.886,A -85,B 0,C 180,E1 -11535.677,E2 -11535.677} C_VEL
LIN {X 0,Y 390.104,Z 499.895,A -85,B 0,C 180,E1 -11538.922,E2 -11538.922} C_VEL
LIN {X 0,Y 390.041,Z 499.899,A -85,B 0,C 180,E1 -11542.234,E2 -11542.234} C_VEL
LIN {X 0,Y 390.085,Z 499.892,A -85,B 0,C 180,E1 -11545.732,E2 -11545.732} C_VEL
LIN {X 0,Y 390.034,Z 499.902,A -85,B 0,C 180,E1 -11549.111,E2 -11549.111} C_VEL
LIN {X 0,Y 390.044,Z 499.902,A -85,B 0,C 180,E1 -11552.721,E2 -11552.721} C_VEL
LIN {X 0,Y 390.056,Z 499.896,A -85,B 0,C 180,E1 -11555.825,E2 -11555.825} C_VEL
LIN {X 0,Y 390.067,Z 499.897,A -85,B 0,C 180,E1 -11559.218,E2 -11559.218} C_VEL
LIN {X 0,Y 390.043,Z 499.9,A -85,B 0,C 180,E1 -11562.374,E2 -11562.374} C_VEL
LIN {X 0,Y 390.093,Z 500.034,A -85,B 0,C 180,E1 -11565.578,E2 -11565.578} C_VEL
LIN {X 0,Y 392.178,Z 510.502,A -85,B 0,C 180,E1 -11569.358,E2 -11569.358} C_VEL
LIN {X 0,Y 393.816,Z 518.898,A -85,B 0,C 180,E1 -11572.232,E2 -11572.232} C_VEL
LIN {X 0,Y 393.84,Z 522.611,A -85,B 0,C 180,E1 -11573.419,E2 -11573.419} C_VEL
LIN {X 0,Y 392.747,Z 533.79,A -85,B 0,C 180,E1 -11576.849,E2 -11576.849} C_VEL
LIN {X 0,Y 391.956,Z 543.857,A -85,B 0,C 180,E1 -11579.864,E2 -11579.864} C_VEL
LIN {X 0,Y 390.918,Z 558.036,A -85,B 0,C 180,E1 -11584.015,E2 -11584.015} C_VEL
LIN {X 0,Y 390.292,Z 569.237,A -85,B 0,C 180,E1 -11587.223,E2 -11587.223} C_VEL
LIN {X 0,Y 389.783,Z 580.831,A -85,B 0,C 180,E1 -11590.515,E2 -11590.515} C_VEL
LIN {X 0,Y 389.625,Z 584.994,A -85,B 0,C 180,E1 -11591.656,E2 -11591.656} C_VEL
LIN {X 0,Y 391.179,Z 599.153,A -85,B 0,C 180,E1 -11592.162,E2 -11592.162} C_VEL
LIN {X 0,Y 392.131,Z 612.351,A -85,B 0,C 180,E1 -11592.83,E2 -11592.83} C_VEL
LIN {X 0,Y 392.716,Z 624.257,A -85,B 0,C 180,E1 -11593.629,E2 -11593.629} C_VEL
LIN {X 0,Y 392.408,Z 632.484,A -85,B 0,C 180,E1 -11594.283,E2 -11594.283} C_VEL
LIN {X 0,Y 391.536,Z 643.174,A -85,B 0,C 180,E1 -11595.313,E2 -11595.313} C_VEL
LIN {X 0,Y 390.618,Z 652.95,A -85,B 0,C 180,E1 -11596.474,E2 -11596.474} C_VEL
LIN {X 0,Y 390.421,Z 658.59,A -85,B 0,C 180,E1 -11597.261,E2 -11597.261} C_VEL
LIN {X 0,Y 389.849,Z 666.586,A -85,B 0,C 180,E1 -11598.562,E2 -11598.562} C_VEL
LIN {X 0,Y 389.452,Z 674.425,A -85,B 0,C 180,E1 -11600.129,E2 -11600.129} C_VEL
LIN {X 0,Y 389.294,Z 680.719,A -85,B 0,C 180,E1 -11601.696,E2 -11601.696} C_VEL
LIN {X 0,Y 389.235,Z 685.688,A -85,B 0,C 180,E1 -11603.255,E2 -11603.255} C_VEL
LIN {X 0,Y 389.393,Z 689.537,A -85,B 0,C 180,E1 -11604.823,E2 -11604.823} C_VEL
LIN {X 0,Y 389.504,Z 691.494,A -85,B 0,C 180,E1 -11605.861,E2 -11605.861} C_VEL
LIN {X 0,Y 389.468,Z 692.988,A -85,B 0,C 180,E1 -11606.897,E2 -11606.897} C_VEL
LIN {X 0,Y 389.506,Z 694.014,A -85,B 0,C 180,E1 -11607.932,E2 -11607.932} C_VEL
LIN {X 0,Y 389.772,Z 694.844,A -85,B 0,C 180,E1 -11610,E2 -11610} C_VEL
LIN {X 0,Y 389.558,Z 694.587,A -85,B 0,C 180,E1 -11611.034,E2 -11611.034} C_VEL
LIN {X 0,Y 389.517,Z 693.894,A -85,B 0,C 180,E1 -11612.068,E2 -11612.068} C_VEL
LIN {X 0,Y 389.533,Z 691.275,A -85,B 0,C 180,E1 -11614.139,E2 -11614.139} C_VEL
LIN {X 0,Y 389.304,Z 688.091,A -85,B 0,C 180,E1 -11615.698,E2 -11615.698} C_VEL
LIN {X 0,Y 389.254,Z 683.85,A -85,B 0,C 180,E1 -11617.261,E2 -11617.261} C_VEL
LIN {X 0,Y 389.341,Z 677.422,A -85,B 0,C 180,E1 -11619.088,E2 -11619.088} C_VEL
LIN {X 0,Y 389.592,Z 670.43,A -85,B 0,C 180,E1 -11620.656,E2 -11620.656} C_VEL
LIN {X 0,Y 390.071,Z 661.83,A -85,B 0,C 180,E1 -11622.222,E2 -11622.222} C_VEL
LIN {X 0,Y 390.597,Z 654.998,A -85,B 0,C 180,E1 -11623.263,E2 -11623.263} C_VEL
LIN {X 0,Y 391.301,Z 646.063,A -85,B 0,C 180,E1 -11624.418,E2 -11624.418} C_VEL
LIN {X 0,Y 392.273,Z 635.063,A -85,B 0,C 180,E1 -11625.59,E2 -11625.59} C_VEL
LIN {X 0,Y 392.998,Z 626.264,A -85,B 0,C 180,E1 -11626.359,E2 -11626.359} C_VEL
LIN {X 0,Y 392.589,Z 615.528,A -85,B 0,C 180,E1 -11627.18,E2 -11627.18} C_VEL
LIN {X 0,Y 392.171,Z 603.148,A -85,B 0,C 180,E1 -11627.932,E2 -11627.932} C_VEL
LIN {X 0,Y 391.031,Z 590.027,A -85,B 0,C 180,E1 -11628.553,E2 -11628.553} C_VEL
LIN {X 0,Y 389.631,Z 579.935,A -85,B 0,C 180,E1 -11628.946,E2 -11628.946} C_VEL
LIN {X 0,Y 389.995,Z 567.994,A -85,B 0,C 180,E1 -11632.237,E2 -11632.237} C_VEL
LIN {X 0,Y 390.617,Z 554.992,A -85,B 0,C 180,E1 -11635.894,E2 -11635.894} C_VEL
LIN {X 0,Y 391.327,Z 542.263,A -85,B 0,C 180,E1 -11639.596,E2 -11639.596} C_VEL
LIN {X 0,Y 392.239,Z 530.603,A -85,B 0,C 180,E1 -11643.126,E2 -11643.126} C_VEL
LIN {X 0,Y 393.236,Z 520.085,A -85,B 0,C 180,E1 -11646.462,E2 -11646.462} C_VEL
LIN {X 0,Y 393.219,Z 516.25,A -85,B 0,C 180,E1 -11647.761,E2 -11647.761} C_VEL
LIN {X 0,Y 391.858,Z 508.523,A -85,B 0,C 180,E1 -11650.634,E2 -11650.634} C_VEL
LIN {X 0,Y 390.097,Z 499.946,A -85,B 0,C 180,E1 -11654.177,E2 -11654.177} C_VEL
LIN {X 0,Y 390.045,Z 499.906,A -85,B 0,C 180,E1 -11657.626,E2 -11657.626} C_VEL
LIN {X 0,Y 390.092,Z 499.897,A -85,B 0,C 180,E1 -11660.908,E2 -11660.908} C_VEL
LIN {X 0,Y 390.087,Z 499.897,A -85,B 0,C 180,E1 -11664.793,E2 -11664.793} C_VEL
LIN {X 0,Y 390.026,Z 499.899,A -85,B 0,C 180,E1 -11668.496,E2 -11668.496} C_VEL
LIN {X 0,Y 390.12,Z 499.89,A -85,B 0,C 180,E1 -11672.07,E2 -11672.07} C_VEL
LIN {X 0,Y 390.083,Z 499.892,A -85,B 0,C 180,E1 -11675.52,E2 -11675.52} C_VEL
LIN {X 0,Y 390.059,Z 499.893,A -85,B 0,C 180,E1 -11678.878,E2 -11678.878} C_VEL
LIN {X 0,Y 390.131,Z 499.885,A -85,B 0,C 180,E1 -11682.167,E2 -11682.167} C_VEL
LIN {X 0,Y 390.148,Z 499.882,A -85,B 0,C 180,E1 -11685.393,E2 -11685.393} C_VEL
LIN {X 0,Y 390.151,Z 499.883,A -85,B 0,C 180,E1 -11688.571,E2 -11688.571} C_VEL
LIN {X 0,Y 390.348,Z 499.857,A -85,B 0,C 180,E1 -11691.993,E2 -11691.993} C_VEL
LIN {X 0,Y 390.226,Z 499.873,A -85,B 0,C 180,E1 -11694.834,E2 -11694.834} C_VEL
LIN {X 0,Y 390.417,Z 499.852,A -85,B 0,C 180,E1 -11697.937,E2 -11697.937} C_VEL
LIN {X 0,Y 390.55,Z 499.837,A -85,B 0,C 180,E1 -11700,E2 -11700} C_VEL
LIN {X 0,Y 390.313,Z 499.868,A -85,B 0,C 180,E1 -11703.097,E2 -11703.097} C_VEL
LIN {X 0,Y 390.266,Z 499.868,A -85,B 0,C 180,E1 -11706.518,E2 -11706.518} C_VEL
LIN {X 0,Y 390.208,Z 499.878,A -85,B 0,C 180,E1 -11709.329,E2 -11709.329} C_VEL
LIN {X 0,Y 390.199,Z 499.88,A -85,B 0,C 180,E1 -11713.439,E2 -11713.439} C_VEL
LIN {X 0,Y 390.171,Z 500.069,A -85,B 0,C 180,E1 -11715.978,E2 -11715.978} C_VEL
LIN {X 0,Y 394.123,Z 511.707,A -85,B 0,C 180,E1 -11716.978,E2 -11716.978} C_VEL
LIN {X 0,Y 396.138,Z 519.035,A -85,B 0,C 180,E1 -11717.688,E2 -11717.688} C_VEL
LIN {X 0,Y 395.402,Z 529.57,A -85,B 0,C 180,E1 -11718.66,E2 -11718.66} C_VEL
LIN {X 0,Y 394.558,Z 540.439,A -85,B 0,C 180,E1 -11719.918,E2 -11719.918} C_VEL
LIN {X 0,Y 393.755,Z 548.817,A -85,B 0,C 180,E1 -11721.111,E2 -11721.111} C_VEL
LIN {X 0,Y 392.866,Z 557.389,A -85,B 0,C 180,E1 -11722.62,E2 -11722.62} C_VEL
LIN {X 0,Y 392.067,Z 565.152,A -85,B 0,C 180,E1 -11724.349,E2 -11724.349} C_VEL
LIN {X 0,Y 391.386,Z 571.281,A -85,B 0,C 180,E1 -11726.124,E2 -11726.124} C_VEL
LIN {X 0,Y 390.872,Z 575.808,A -85,B 0,C 180,E1 -11727.872,E2 -11727.872} C_VEL
LIN {X 0,Y 390.597,Z 578.16,A -85,B 0,C 180,E1 -11729.066,E2 -11729.066} C_VEL
LIN {X 0,Y 390.338,Z 579.913,A -85,B 0,C 180,E1 -11730.275,E2 -11730.275} C_VEL
LIN {X 0,Y 390.076,Z 581.559,A -85,B 0,C 180,E1 -11732.134,E2 -11732.134} C_VEL
LIN {X 0,Y 389.966,Z 581.905,A -85,B 0,C 180,E1 -11734.002,E2 -11734.002} C_VEL
LIN {X 0,Y 389.975,Z 580.998,A -85,B 0,C 180,E1 -11735.808,E2 -11735.808} C_VEL
LIN {X 0,Y 390.082,Z 578.642,A -85,B 0,C 180,E1 -11737.776,E2 -11737.776} C_VEL
LIN {X 0,Y 390.396,Z 574.684,A -85,B 0,C 180,E1 -11739.77,E2 -11739.77} C_VEL
LIN {X 0,Y 390.84,Z 569.176,A -85,B 0,C 180,E1 -11741.708,E2 -11741.708} C_VEL
LIN {X 0,Y 391.33,Z 563.197,A -85,B 0,C 180,E1 -11743.315,E2 -11743.315} C_VEL
LIN {X 0,Y 391.872,Z 556.579,A -85,B 0,C 180,E1 -11744.744,E2 -11744.744} C_VEL
LIN {X 0,Y 392.608,Z 547.764,A -85,B 0,C 180,E1 -11746.282,E2 -11746.282} C_VEL
LIN {X 0,Y 393.296,Z 537.93,A -85,B 0,C 180,E1 -11747.676,E2 -11747.676} C_VEL
LIN {X 0,Y 393.984,Z 527.18,A -85,B 0,C 180,E1 -11748.893,E2 -11748.893} C_VEL
LIN {X 0,Y 394.632,Z 516.974,A -85,B 0,C 180,E1 -11749.824,E2 -11749.824} C_VEL
LIN {X 0,Y 393.829,Z 513.013,A -85,B 0,C 180,E1 -11750.185,E2 -11750.185} C_VEL
LIN {X 0,Y 390.538,Z 501.615,A -85,B 0,C 180,E1 -11751.126,E2 -11751.126} C_VEL
LIN {X 0,Y 390.075,Z 499.898,A -85,B 0,C 180,E1 -11751.279,E2 -11751.279} C_VEL
LIN {X 0,Y 390.09,Z 499.893,A -85,B 0,C 180,E1 -11754.793,E2 -11754.793} C_VEL
LIN {X 0,Y 390.029,Z 499.9,A -85,B 0,C 180,E1 -11758.496,E2 -11758.496} C_VEL
LIN {X 0,Y 390.122,Z 499.888,A -85,B 0,C 180,E1 -11762.07,E2 -11762.07} C_VEL
LIN {X 0,Y 390.08,Z 499.897,A -85,B 0,C 180,E1 -11765.519,E2 -11765.519} C_VEL
LIN {X 0,Y 390.093,Z 499.895,A -85,B 0,C 180,E1 -11769.53,E2 -11769.53} C_VEL
LIN {X 0,Y 390.143,Z 499.889,A -85,B 0,C 180,E1 -11773.248,E2 -11773.248} C_VEL
LIN {X 0,Y 390.2,Z 499.879,A -85,B 0,C 180,E1 -11776.562,E2 -11776.562} C_VEL
LIN {X 0,Y 390.173,Z 499.884,A -85,B 0,C 180,E1 -11779.623,E2 -11779.623} C_VEL
LIN {X 0,Y 390.253,Z 499.873,A -85,B 0,C 180,E1 -11782.758,E2 -11782.758} C_VEL
LIN {X 0,Y 390.219,Z 499.877,A -85,B 0,C 180,E1 -11784.833,E2 -11784.833} C_VEL
LIN {X 0,Y 390.423,Z 499.852,A -85,B 0,C 180,E1 -11787.937,E2 -11787.937} C_VEL
LIN {X 0,Y 390.545,Z 499.836,A -85,B 0,C 180,E1 -11790,E2 -11790} C_VEL
LIN {X 0,Y 390.306,Z 499.87,A -85,B 0,C 180,E1 -11793.096,E2 -11793.096} C_VEL
LIN {X 0,Y 390.291,Z 499.867,A -85,B 0,C 180,E1 -11796.202,E2 -11796.202} C_VEL
LIN {X 0,Y 390.198,Z 499.882,A -85,B 0,C 180,E1 -11799.329,E2 -11799.329} C_VEL
LIN {X 0,Y 390.176,Z 499.882,A -85,B 0,C 180,E1 -11802.483,E2 -11802.483} C_VEL
LIN {X 0,Y 390.144,Z 499.888,A -85,B 0,C 180,E1 -11805.677,E2 -11805.677} C_VEL
LIN {X 0,Y 390.107,Z 499.892,A -85,B 0,C 180,E1 -11808.922,E2 -11808.922} C_VEL
LIN {X 0,Y 390.044,Z 499.898,A -85,B 0,C 180,E1 -11812.234,E2 -11812.234} C_VEL
LIN {X 0,Y 390.059,Z 499.895,A -85,B 0,C 180,E1 -11814.151,E2 -11814.151} C_VEL
LIN {X 0,Y 389.406,Z 499.98,A -85,B 0,C 180,E1 -11815.012,E2 -11815.012} C_VEL
LIN {X 0,Y 386.57,Z 500.334,A -85,B 0,C 180,E1 -11816.413,E2 -11816.413} C_VEL
LIN {X 0,Y 384.148,Z 500.636,A -85,B 0,C 180,E1 -11817.545,E2 -11817.545} C_VEL
LIN {X 0,Y 383.087,Z 500.765,A -85,B 0,C 180,E1 -11818.421,E2 -11818.421} C_VEL
LIN {X 0,Y 382.99,Z 500.776,A -85,B 0,C 180,E1 -11818.717,E2 -11818.717} C_VEL
LIN {X 0,Y 383.013,Z 500.773,A -85,B 0,C 180,E1 -11822.149,E2 -11822.149} C_VEL
LIN {X 0,Y 383.021,Z 500.775,A -85,B 0,C 180,E1 -11824.668,E2 -11824.668} C_VEL
LIN {X 0,Y 382.998,Z 500.775,A -85,B 0,C 180,E1 -11827.902,E2 -11827.902} C_VEL
LIN {X 0,Y 382.965,Z 500.784,A -85,B 0,C 180,E1 -11831.35,E2 -11831.35} C_VEL
LIN {X 0,Y 382.997,Z 500.775,A -85,B 0,C 180,E1 -11834.303,E2 -11834.303} C_VEL
LIN {X 0,Y 383.013,Z 500.778,A -85,B 0,C 180,E1 -11837.24,E2 -11837.24} C_VEL
LIN {X 0,Y 383.013,Z 500.774,A -85,B 0,C 180,E1 -11840.414,E2 -11840.414} C_VEL
LIN {X 0,Y 383.027,Z 500.772,A -85,B 0,C 180,E1 -11844.044,E2 -11844.044} C_VEL
LIN {X 0,Y 382.99,Z 500.778,A -85,B 0,C 180,E1 -11847.578,E2 -11847.578} C_VEL
LIN {X 0,Y 382.995,Z 500.776,A -85,B 0,C 180,E1 -11850.3,E2 -11850.3} C_VEL
LIN {X 0,Y 383.082,Z 500.765,A -85,B 0,C 180,E1 -11854.021,E2 -11854.021} C_VEL
LIN {X 0,Y 382.994,Z 500.778,A -85,B 0,C 180,E1 -11857.334,E2 -11857.334} C_VEL
LIN {X 0,Y 383.063,Z 500.771,A -85,B 0,C 180,E1 -11860.716,E2 -11860.716} C_VEL
LIN {X 0,Y 383.083,Z 500.764,A -85,B 0,C 180,E1 -11864.026,E2 -11864.026} C_VEL
LIN {X 0,Y 383.139,Z 500.761,A -85,B 0,C 180,E1 -11867.284,E2 -11867.284} C_VEL
LIN {X 0,Y 383.146,Z 500.758,A -85,B 0,C 180,E1 -11870.497,E2 -11870.497} C_VEL
LIN {X 0,Y 383.257,Z 500.743,A -85,B 0,C 180,E1 -11873.683,E2 -11873.683} C_VEL
LIN {X 0,Y 383.385,Z 500.727,A -85,B 0,C 180,E1 -11877.899,E2 -11877.899} C_VEL
LIN {X 0,Y 383.516,Z 500.711,A -85,B 0,C 180,E1 -11880,E2 -11880} C_VEL
LIN {X 0,Y 383.211,Z 500.752,A -85,B 0,C 180,E1 -11883.154,E2 -11883.154} C_VEL
LIN {X 0,Y 383.244,Z 500.746,A -85,B 0,C 180,E1 -11886.317,E2 -11886.317} C_VEL
LIN {X 0,Y 383.154,Z 500.757,A -85,B 0,C 180,E1 -11889.502,E2 -11889.502} C_VEL
LIN {X 0,Y 383.143,Z 500.761,A -85,B 0,C 180,E1 -11892.716,E2 -11892.716} C_VEL
LIN {X 0,Y 383.082,Z 500.765,A -85,B 0,C 180,E1 -11895.973,E2 -11895.973} C_VEL
LIN {X 0,Y 383.06,Z 500.769,A -85,B 0,C 180,E1 -11899.284,E2 -11899.284} C_VEL
LIN {X 0,Y 382.998,Z 500.779,A -85,B 0,C 180,E1 -11902.665,E2 -11902.665} C_VEL
LIN {X 0,Y 383.014,Z 500.773,A -85,B 0,C 180,E1 -11906.128,E2 -11906.128} C_VEL
LIN {X 0,Y 382.981,Z 500.778,A -85,B 0,C 180,E1 -11909.701,E2 -11909.701} C_VEL
LIN {X 0,Y 383.004,Z 500.776,A -85,B 0,C 180,E1 -11913.401,E2 -11913.401} C_VEL
LIN {X 0,Y 383.032,Z 500.772,A -85,B 0,C 180,E1 -11916.164,E2 -11916.164} C_VEL
LIN {X 0,Y 383.008,Z 500.778,A -85,B 0,C 180,E1 -11919.958,E2 -11919.958} C_VEL
LIN {X 0,Y 383.006,Z 500.779,A -85,B 0,C 180,E1 -11922.778,E2 -11922.778} C_VEL
LIN {X 0,Y 383.027,Z 500.858,A -85,B 0,C 180,E1 -11925.226,E2 -11925.226} C_VEL
LIN {X 0,Y 385.03,Z 510.889,A -85,B 0,C 180,E1 -11928.92,E2 -11928.92} C_VEL
LIN {X 0,Y 386.862,Z 520.204,A -85,B 0,C 180,E1 -11932.18,E2 -11932.18} C_VEL
LIN {X 0,Y 386.903,Z 523.222,A -85,B 0,C 180,E1 -11933.17,E2 -11933.17} C_VEL
LIN {X 0,Y 385.891,Z 533.07,A -85,B 0,C 180,E1 -11936.256,E2 -11936.256} C_VEL
LIN {X 0,Y 385.081,Z 542.893,A -85,B 0,C 180,E1 -11939.268,E2 -11939.268} C_VEL
LIN {X 0,Y 383.988,Z 556.439,A -85,B 0,C 180,E1 -11943.328,E2 -11943.328} C_VEL
LIN {X 0,Y 383.267,Z 568.56,A -85,B 0,C 180,E1 -11946.891,E2 -11946.891} C_VEL
LIN {X 0,Y 382.664,Z 581.694,A -85,B 0,C 180,E1 -11950.696,E2 -11950.696} C_VEL
LIN {X 0,Y 382.558,Z 584.09,A -85,B 0,C 180,E1 -11951.351,E2 -11951.351} C_VEL
LIN {X 0,Y 384.132,Z 598.419,A -85,B 0,C 180,E1 -11951.879,E2 -11951.879} C_VEL
LIN {X 0,Y 385.059,Z 611.427,A -85,B 0,C 180,E1 -11952.555,E2 -11952.555} C_VEL
LIN {X 0,Y 385.671,Z 624.435,A -85,B 0,C 180,E1 -11953.457,E2 -11953.457} C_VEL
LIN {X 0,Y 385.407,Z 632.475,A -85,B 0,C 180,E1 -11954.126,E2 -11954.126} C_VEL
LIN {X 0,Y 384.517,Z 642.972,A -85,B 0,C 180,E1 -11955.174,E2 -11955.174} C_VEL
LIN {X 0,Y 383.542,Z 653.601,A -85,B 0,C 180,E1 -11956.489,E2 -11956.489} C_VEL
LIN {X 0,Y 383.09,Z 660.672,A -85,B 0,C 180,E1 -11957.552,E2 -11957.552} C_VEL
LIN {X 0,Y 382.586,Z 669.519,A -85,B 0,C 180,E1 -11959.147,E2 -11959.147} C_VEL
LIN {X 0,Y 382.275,Z 676.58,A -85,B 0,C 180,E1 -11960.743,E2 -11960.743} C_VEL
LIN {X 0,Y 382.174,Z 683.057,A -85,B 0,C 180,E1 -11962.604,E2 -11962.604} C_VEL
LIN {X 0,Y 382.231,Z 687.286,A -85,B 0,C 180,E1 -11964.196,E2 -11964.196} C_VEL
LIN {X 0,Y 382.466,Z 690.422,A -85,B 0,C 180,E1 -11965.785,E2 -11965.785} C_VEL
LIN {X 0,Y 382.432,Z 691.927,A -85,B 0,C 180,E1 -11966.84,E2 -11966.84} C_VEL
LIN {X 0,Y 382.471,Z 692.968,A -85,B 0,C 180,E1 -11967.894,E2 -11967.894} C_VEL
LIN {X 0,Y 382.748,Z 693.813,A -85,B 0,C 180,E1 -11970,E2 -11970} C_VEL
LIN {X 0,Y 382.527,Z 693.562,A -85,B 0,C 180,E1 -11971.053,E2 -11971.053} C_VEL
LIN {X 0,Y 382.477,Z 692.88,A -85,B 0,C 180,E1 -11972.106,E2 -11972.106} C_VEL
LIN {X 0,Y 382.441,Z 691.777,A -85,B 0,C 180,E1 -11973.16,E2 -11973.16} C_VEL
LIN {X 0,Y 382.47,Z 690.263,A -85,B 0,C 180,E1 -11974.215,E2 -11974.215} C_VEL
LIN {X 0,Y 382.241,Z 687.089,A -85,B 0,C 180,E1 -11975.804,E2 -11975.804} C_VEL
LIN {X 0,Y 382.191,Z 682.856,A -85,B 0,C 180,E1 -11977.396,E2 -11977.396} C_VEL
LIN {X 0,Y 382.254,Z 677.456,A -85,B 0,C 180,E1 -11978.991,E2 -11978.991} C_VEL
LIN {X 0,Y 382.465,Z 670.745,A -85,B 0,C 180,E1 -11980.589,E2 -11980.589} C_VEL
LIN {X 0,Y 382.974,Z 662.464,A -85,B 0,C 180,E1 -11982.183,E2 -11982.183} C_VEL
LIN {X 0,Y 383.54,Z 654.114,A -85,B 0,C 180,E1 -11983.511,E2 -11983.511} C_VEL
LIN {X 0,Y 384.593,Z 642.965,A -85,B 0,C 180,E1 -11984.959,E2 -11984.959} C_VEL
LIN {X 0,Y 385.663,Z 631.606,A -85,B 0,C 180,E1 -11986.135,E2 -11986.135} C_VEL
LIN {X 0,Y 385.959,Z 625.616,A -85,B 0,C 180,E1 -11986.666,E2 -11986.666} C_VEL
LIN {X 0,Y 385.683,Z 613.148,A -85,B 0,C 180,E1 -11987.628,E2 -11987.628} C_VEL
LIN {X 0,Y 385.152,Z 600.33,A -85,B 0,C 180,E1 -11988.402,E2 -11988.402} C_VEL
LIN {X 0,Y 383.737,Z 586.379,A -85,B 0,C 180,E1 -11989.059,E2 -11989.059} C_VEL
LIN {X 0,Y 382.613,Z 578.687,A -85,B 0,C 180,E1 -11989.377,E2 -11989.377} C_VEL
LIN {X 0,Y 383.022,Z 565.634,A -85,B 0,C 180,E1 -11993.067,E2 -11993.067} C_VEL
LIN {X 0,Y 383.697,Z 553.204,A -85,B 0,C 180,E1 -11996.664,E2 -11996.664} C_VEL
LIN {X 0,Y 384.447,Z 541.445,A -85,B 0,C 180,E1 -12000.181,E2 -12000.181} C_VEL
LIN {X 0,Y 385.381,Z 529.857,A -85,B 0,C 180,E1 -12003.795,E2 -12003.795} C_VEL
LIN {X 0,Y 386.384,Z 520.396,A -85,B 0,C 180,E1 -12006.888,E2 -12006.888} C_VEL
LIN {X 0,Y 386.121,Z 516.601,A -85,B 0,C 180,E1 -12008.233,E2 -12008.233} C_VEL
LIN {X 0,Y 384.575,Z 508.249,A -85,B 0,C 180,E1 -12011.473,E2 -12011.473} C_VEL
LIN {X 0,Y 383.038,Z 500.779,A -85,B 0,C 180,E1 -12014.729,E2 -12014.729} C_VEL
LIN {X 0,Y 383.012,Z 500.781,A -85,B 0,C 180,E1 -12017.24,E2 -12017.24} C_VEL
LIN {X 0,Y 383.017,Z 500.777,A -85,B 0,C 180,E1 -12020.414,E2 -12020.414} C_VEL
LIN {X 0,Y 383.027,Z 500.773,A -85,B 0,C 180,E1 -12024.045,E2 -12024.045} C_VEL
LIN {X 0,Y 382.989,Z 500.777,A -85,B 0,C 180,E1 -12027.578,E2 -12027.578} C_VEL
LIN {X 0,Y 382.995,Z 500.774,A -85,B 0,C 180,E1 -12030.3,E2 -12030.3} C_VEL
LIN {X 0,Y 383.059,Z 500.766,A -85,B 0,C 180,E1 -12032.698,E2 -12032.698} C_VEL
LIN {X 0,Y 383.036,Z 500.768,A -85,B 0,C 180,E1 -12036.193,E2 -12036.193} C_VEL
LIN {X 0,Y 383.059,Z 500.766,A -85,B 0,C 180,E1 -12039.599,E2 -12039.599} C_VEL
LIN {X 0,Y 383.108,Z 500.763,A -85,B 0,C 180,E1 -12042.932,E2 -12042.932} C_VEL
LIN {X 0,Y 383.129,Z 500.762,A -85,B 0,C 180,E1 -12046.464,E2 -12046.464} C_VEL
LIN {X 0,Y 383.155,Z 500.759,A -85,B 0,C 180,E1 -12050.498,E2 -12050.498} C_VEL
LIN {X 0,Y 383.278,Z 500.741,A -85,B 0,C 180,E1 -12052.626,E2 -12052.626} C_VEL
LIN {X 0,Y 383.199,Z 500.749,A -85,B 0,C 180,E1 -12054.739,E2 -12054.739} C_VEL
LIN {X 0,Y 383.383,Z 500.729,A -85,B 0,C 180,E1 -12057.899,E2 -12057.899} C_VEL
LIN {X 0,Y 383.52,Z 500.713,A -85,B 0,C 180,E1 -12060,E2 -12060} C_VEL
LIN {X 0,Y 383.249,Z 500.749,A -85,B 0,C 180,E1 -12063.154,E2 -12063.154} C_VEL
LIN {X 0,Y 383.23,Z 500.745,A -85,B 0,C 180,E1 -12066.506,E2 -12066.506} C_VEL
LIN {X 0,Y 383.155,Z 500.757,A -85,B 0,C 180,E1 -12069.502,E2 -12069.502} C_VEL
LIN {X 0,Y 383.13,Z 500.761,A -85,B 0,C 180,E1 -12073.536,E2 -12073.536} C_VEL
LIN {X 0,Y 383.119,Z 500.766,A -85,B 0,C 180,E1 -12075.528,E2 -12075.528} C_VEL
LIN {X 0,Y 387.642,Z 514.076,A -85,B 0,C 180,E1 -12076.728,E2 -12076.728} C_VEL
LIN {X 0,Y 389.411,Z 519.948,A -85,B 0,C 180,E1 -12077.325,E2 -12077.325} C_VEL
LIN {X 0,Y 388.685,Z 531.654,A -85,B 0,C 180,E1 -12078.447,E2 -12078.447} C_VEL
LIN {X 0,Y 387.866,Z 541.129,A -85,B 0,C 180,E1 -12079.57,E2 -12079.57} C_VEL
LIN {X 0,Y 387.079,Z 549.225,A -85,B 0,C 180,E1 -12080.736,E2 -12080.736} C_VEL
LIN {X 0,Y 386.2,Z 557.192,A -85,B 0,C 180,E1 -12082.12,E2 -12082.12} C_VEL
LIN {X 0,Y 385.46,Z 564.274,A -85,B 0,C 180,E1 -12083.649,E2 -12083.649} C_VEL
LIN {X 0,Y 384.689,Z 570.767,A -85,B 0,C 180,E1 -12085.425,E2 -12085.425} C_VEL
LIN {X 0,Y 384.059,Z 575.787,A -85,B 0,C 180,E1 -12087.225,E2 -12087.225} C_VEL
LIN {X 0,Y 383.75,Z 578.383,A -85,B 0,C 180,E1 -12088.468,E2 -12088.468} C_VEL
LIN {X 0,Y 383.313,Z 581.365,A -85,B 0,C 180,E1 -12090.487,E2 -12090.487} C_VEL
LIN {X 0,Y 383.046,Z 582.769,A -85,B 0,C 180,E1 -12092.435,E2 -12092.435} C_VEL
LIN {X 0,Y 382.936,Z 582.849,A -85,B 0,C 180,E1 -12094.321,E2 -12094.321} C_VEL
LIN {X 0,Y 382.959,Z 581.727,A -85,B 0,C 180,E1 -12096.149,E2 -12096.149} C_VEL
LIN {X 0,Y 383.069,Z 579.497,A -85,B 0,C 180,E1 -12097.916,E2 -12097.916} C_VEL
LIN {X 0,Y 383.414,Z 575.51,A -85,B 0,C 180,E1 -12099.908,E2 -12099.908} C_VEL
LIN {X 0,Y 383.885,Z 569.785,A -85,B 0,C 180,E1 -12101.93,E2 -12101.93} C_VEL
LIN {X 0,Y 384.414,Z 563.034,A -85,B 0,C 180,E1 -12103.714,E2 -12103.714} C_VEL
LIN {X 0,Y 385.146,Z 555.094,A -85,B 0,C 180,E1 -12105.371,E2 -12105.371} C_VEL
LIN {X 0,Y 385.812,Z 546.79,A -85,B 0,C 180,E1 -12106.774,E2 -12106.774} C_VEL
LIN {X 0,Y 386.604,Z 536.401,A -85,B 0,C 180,E1 -12108.188,E2 -12108.188} C_VEL
LIN {X 0,Y 387.3,Z 526.039,A -85,B 0,C 180,E1 -12109.332,E2 -12109.332} C_VEL
LIN {X 0,Y 387.774,Z 518.516,A -85,B 0,C 180,E1 -12110.017,E2 -12110.017} C_VEL
LIN {X 0,Y 386.282,Z 512.07,A -85,B 0,C 180,E1 -12110.616,E2 -12110.616} C_VEL
LIN {X 0,Y 383.025,Z 500.775,A -85,B 0,C 180,E1 -12111.549,E2 -12111.549} C_VEL
LIN {X 0,Y 383.029,Z 500.772,A -85,B 0,C 180,E1 -12114.045,E2 -12114.045} C_VEL
LIN {X 0,Y 382.992,Z 500.779,A -85,B 0,C 180,E1 -12117.578,E2 -12117.578} C_VEL
LIN {X 0,Y 382.997,Z 500.775,A -85,B 0,C 180,E1 -12120.3,E2 -12120.3} C_VEL
LIN {X 0,Y 383.061,Z 500.768,A -85,B 0,C 180,E1 -12122.698,E2 -12122.698} C_VEL
LIN {X 0,Y 383.054,Z 500.772,A -85,B 0,C 180,E1 -12125.04,E2 -12125.04} C_VEL
LIN {X 0,Y 382.997,Z 500.775,A -85,B 0,C 180,E1 -12128.469,E2 -12128.469} C_VEL
LIN {X 0,Y 383.058,Z 500.77,A -85,B 0,C 180,E1 -12131.826,E2 -12131.826} C_VEL
LIN {X 0,Y 383.115,Z 500.765,A -85,B 0,C 180,E1 -12135.118,E2 -12135.118} C_VEL
LIN {X 0,Y 383.102,Z 500.762,A -85,B 0,C 180,E1 -12138.358,E2 -12138.358} C_VEL
LIN {X 0,Y 383.22,Z 500.748,A -85,B 0,C 180,E1 -12142.028,E2 -12142.028} C_VEL
LIN {X 0,Y 383.19,Z 500.753,A -85,B 0,C 180,E1 -12144.738,E2 -12144.738} C_VEL
LIN {X 0,Y 383.39,Z 500.728,A -85,B 0,C 180,E1 -12147.899,E2 -12147.899} C_VEL
LIN {X 0,Y 383.515,Z 500.711,A -85,B 0,C 180,E1 -12150,E2 -12150} C_VEL
LIN {X 0,Y 383.242,Z 500.749,A -85,B 0,C 180,E1 -12153.154,E2 -12153.154} C_VEL
LIN {X 0,Y 383.247,Z 500.744,A -85,B 0,C 180,E1 -12156.317,E2 -12156.317} C_VEL
LIN {X 0,Y 383.148,Z 500.76,A -85,B 0,C 180,E1 -12159.502,E2 -12159.502} C_VEL
LIN {X 0,Y 383.13,Z 500.761,A -85,B 0,C 180,E1 -12163.536,E2 -12163.536} C_VEL
LIN {X 0,Y 383.099,Z 500.766,A -85,B 0,C 180,E1 -12167.069,E2 -12167.069} C_VEL
LIN {X 0,Y 383.033,Z 500.772,A -85,B 0,C 180,E1 -12170.647,E2 -12170.647} C_VEL
LIN {X 0,Y 383.016,Z 500.772,A -85,B 0,C 180,E1 -12174.147,E2 -12174.147} C_VEL
LIN {X 0,Y 383.023,Z 500.776,A -85,B 0,C 180,E1 -12177.305,E2 -12177.305} C_VEL
LIN {X 0,Y 382.99,Z 500.776,A -85,B 0,C 180,E1 -12178.717,E2 -12178.717} C_VEL
LIN {X 0,Y 382.295,Z 500.865,A -85,B 0,C 180,E1 -12179.595,E2 -12179.595} C_VEL
LIN {X 0,Y 379.437,Z 501.222,A -85,B 0,C 180,E1 -12181.023,E2 -12181.023} C_VEL
LIN {X 0,Y 377.039,Z 501.52,A -85,B 0,C 180,E1 -12182.177,E2 -12182.177} C_VEL
LIN {X 0,Y 376.016,Z 501.65,A -85,B 0,C 180,E1 -12183.069,E2 -12183.069} C_VEL
LIN {X 0,Y 375.934,Z 501.654,A -85,B 0,C 180,E1 -12183.371,E2 -12183.371} C_VEL
LIN {X 0,Y 375.956,Z 501.655,A -85,B 0,C 180,E1 -12186.741,E2 -12186.741} C_VEL
LIN {X 0,Y 375.942,Z 501.654,A -85,B 0,C 180,E1 -12189.961,E2 -12189.961} C_VEL
LIN {X 0,Y 375.932,Z 501.656,A -85,B 0,C 180,E1 -12193.766,E2 -12193.766} C_VEL
LIN {X 0,Y 375.937,Z 501.658,A -85,B 0,C 180,E1 -12196.81,E2 -12196.81} C_VEL
LIN {X 0,Y 375.96,Z 501.653,A -85,B 0,C 180,E1 -12200.536,E2 -12200.536} C_VEL
LIN {X 0,Y 375.966,Z 501.653,A -85,B 0,C 180,E1 -12203.495,E2 -12203.495} C_VEL
LIN {X 0,Y 375.963,Z 501.651,A -85,B 0,C 180,E1 -12205.888,E2 -12205.888} C_VEL
LIN {X 0,Y 375.968,Z 501.652,A -85,B 0,C 180,E1 -12209.687,E2 -12209.687} C_VEL
LIN {X 0,Y 376.022,Z 501.647,A -85,B 0,C 180,E1 -12213.348,E2 -12213.348} C_VEL
LIN {X 0,Y 375.981,Z 501.653,A -85,B 0,C 180,E1 -12216.887,E2 -12216.887} C_VEL
LIN {X 0,Y 376,Z 501.648,A -85,B 0,C 180,E1 -12220.339,E2 -12220.339} C_VEL
LIN {X 0,Y 376.031,Z 501.643,A -85,B 0,C 180,E1 -12223.719,E2 -12223.719} C_VEL
LIN {X 0,Y 376.106,Z 501.638,A -85,B 0,C 180,E1 -12227.042,E2 -12227.042} C_VEL
LIN {X 0,Y 376.116,Z 501.633,A -85,B 0,C 180,E1 -12230.318,E2 -12230.318} C_VEL
LIN {X 0,Y 376.215,Z 501.621,A -85,B 0,C 180,E1 -12233.564,E2 -12233.564} C_VEL
LIN {X 0,Y 376.351,Z 501.603,A -85,B 0,C 180,E1 -12237.859,E2 -12237.859} C_VEL
LIN {X 0,Y 376.485,Z 501.586,A -85,B 0,C 180,E1 -12240,E2 -12240} C_VEL
LIN {X 0,Y 376.346,Z 501.603,A -85,B 0,C 180,E1 -12242.14,E2 -12242.14} C_VEL
LIN {X 0,Y 376.203,Z 501.624,A -85,B 0,C 180,E1 -12246.435,E2 -12246.435} C_VEL
LIN {X 0,Y 376.122,Z 501.632,A -85,B 0,C 180,E1 -12249.681,E2 -12249.681} C_VEL
LIN {X 0,Y 376.092,Z 501.635,A -85,B 0,C 180,E1 -12253.658,E2 -12253.658} C_VEL
LIN {X 0,Y 376.034,Z 501.644,A -85,B 0,C 180,E1 -12257.4,E2 -12257.4} C_VEL
LIN {X 0,Y 375.979,Z 501.654,A -85,B 0,C 180,E1 -12260.832,E2 -12260.832} C_VEL
LIN {X 0,Y 375.981,Z 501.651,A -85,B 0,C 180,E1 -12264.282,E2 -12264.282} C_VEL
LIN {X 0,Y 375.935,Z 501.655,A -85,B 0,C 180,E1 -12267.863,E2 -12267.863} C_VEL
LIN {X 0,Y 375.958,Z 501.651,A -85,B 0,C 180,E1 -12271.562,E2 -12271.562} C_VEL
LIN {X 0,Y 375.958,Z 501.653,A -85,B 0,C 180,E1 -12275.415,E2 -12275.415} C_VEL
LIN {X 0,Y 375.973,Z 501.651,A -85,B 0,C 180,E1 -12278.27,E2 -12278.27} C_VEL
LIN {X 0,Y 375.935,Z 501.659,A -85,B 0,C 180,E1 -12281.601,E2 -12281.601} C_VEL
LIN {X 0,Y 375.997,Z 501.727,A -85,B 0,C 180,E1 -12284.874,E2 -12284.874} C_VEL
LIN {X 0,Y 378.035,Z 512.085,A -85,B 0,C 180,E1 -12288.774,E2 -12288.774} C_VEL
LIN {X 0,Y 379.671,Z 520.407,A -85,B 0,C 180,E1 -12291.75,E2 -12291.75} C_VEL
LIN {X 0,Y 379.978,Z 523.14,A -85,B 0,C 180,E1 -12292.686,E2 -12292.686} C_VEL
LIN {X 0,Y 379.109,Z 532.092,A -85,B 0,C 180,E1 -12295.569,E2 -12295.569} C_VEL
LIN {X 0,Y 378.008,Z 543.985,A -85,B 0,C 180,E1 -12299.294,E2 -12299.294} C_VEL
LIN {X 0,Y 376.887,Z 557.793,A -85,B 0,C 180,E1 -12303.519,E2 -12303.519} C_VEL
LIN {X 0,Y 376.179,Z 569.063,A -85,B 0,C 180,E1 -12306.9,E2 -12306.9} C_VEL
LIN {X 0,Y 375.629,Z 580.598,A -85,B 0,C 180,E1 -12310.319,E2 -12310.319} C_VEL
LIN {X 0,Y 375.519,Z 582.982,A -85,B 0,C 180,E1 -12311.024,E2 -12311.024} C_VEL
LIN {X 0,Y 377.117,Z 597.813,A -85,B 0,C 180,E1 -12311.592,E2 -12311.592} C_VEL
LIN {X 0,Y 378.027,Z 610.584,A -85,B 0,C 180,E1 -12312.276,E2 -12312.276} C_VEL
LIN {X 0,Y 378.576,Z 622.829,A -85,B 0,C 180,E1 -12313.138,E2 -12313.138} C_VEL
LIN {X 0,Y 378.624,Z 629.483,A -85,B 0,C 180,E1 -12313.695,E2 -12313.695} C_VEL
LIN {X 0,Y 377.658,Z 640.406,A -85,B 0,C 180,E1 -12314.76,E2 -12314.76} C_VEL
LIN {X 0,Y 376.79,Z 650.331,A -85,B 0,C 180,E1 -12315.967,E2 -12315.967} C_VEL
LIN {X 0,Y 376.121,Z 659.407,A -85,B 0,C 180,E1 -12317.317,E2 -12317.317} C_VEL
LIN {X 0,Y 375.565,Z 668.298,A -85,B 0,C 180,E1 -12318.942,E2 -12318.942} C_VEL
LIN {X 0,Y 375.229,Z 675.409,A -85,B 0,C 180,E1 -12320.568,E2 -12320.568} C_VEL
LIN {X 0,Y 375.116,Z 681.916,A -85,B 0,C 180,E1 -12322.464,E2 -12322.464} C_VEL
LIN {X 0,Y 375.17,Z 686.174,A -85,B 0,C 180,E1 -12324.086,E2 -12324.086} C_VEL
LIN {X 0,Y 375.427,Z 689.338,A -85,B 0,C 180,E1 -12325.706,E2 -12325.706} C_VEL
LIN {X 0,Y 375.396,Z 690.855,A -85,B 0,C 180,E1 -12326.78,E2 -12326.78} C_VEL
LIN {X 0,Y 375.436,Z 691.917,A -85,B 0,C 180,E1 -12327.855,E2 -12327.855} C_VEL
LIN {X 0,Y 375.723,Z 692.778,A -85,B 0,C 180,E1 -12330,E2 -12330} C_VEL
LIN {X 0,Y 375.495,Z 692.534,A -85,B 0,C 180,E1 -12331.073,E2 -12331.073} C_VEL
LIN {X 0,Y 375.437,Z 691.865,A -85,B 0,C 180,E1 -12332.146,E2 -12332.146} C_VEL
LIN {X 0,Y 375.398,Z 690.766,A -85,B 0,C 180,E1 -12333.22,E2 -12333.22} C_VEL
LIN {X 0,Y 375.392,Z 689.25,A -85,B 0,C 180,E1 -12334.295,E2 -12334.295} C_VEL
LIN {X 0,Y 375.182,Z 686.087,A -85,B 0,C 180,E1 -12335.914,E2 -12335.914} C_VEL
LIN {X 0,Y 375.127,Z 681.862,A -85,B 0,C 180,E1 -12337.536,E2 -12337.536} C_VEL
LIN {X 0,Y 375.209,Z 675.489,A -85,B 0,C 180,E1 -12339.433,E2 -12339.433} C_VEL
LIN {X 0,Y 375.512,Z 668.551,A -85,B 0,C 180,E1 -12341.06,E2 -12341.06} C_VEL
LIN {X 0,Y 376.1,Z 660.032,A -85,B 0,C 180,E1 -12342.684,E2 -12342.684} C_VEL
LIN {X 0,Y 376.704,Z 651.421,A -85,B 0,C 180,E1 -12344.036,E2 -12344.036} C_VEL
LIN {X 0,Y 377.796,Z 641.061,A -85,B 0,C 180,E1 -12345.372,E2 -12345.372} C_VEL
LIN {X 0,Y 378.96,Z 629.491,A -85,B 0,C 180,E1 -12346.567,E2 -12346.567} C_VEL
LIN {X 0,Y 378.861,Z 616.691,A -85,B 0,C 180,E1 -12347.669,E2 -12347.669} C_VEL
LIN {X 0,Y 378.541,Z 603.94,A -85,B 0,C 180,E1 -12348.533,E2 -12348.533} C_VEL
LIN {X 0,Y 377.393,Z 590.285,A -85,B 0,C 180,E1 -12349.267,E2 -12349.267} C_VEL
LIN {X 0,Y 375.571,Z 577.452,A -85,B 0,C 180,E1 -12349.825,E2 -12349.825} C_VEL
LIN {X 0,Y 376.052,Z 564.133,A -85,B 0,C 180,E1 -12353.686,E2 -12353.686} C_VEL
LIN {X 0,Y 376.738,Z 552.324,A -85,B 0,C 180,E1 -12357.197,E2 -12357.197} C_VEL
LIN {X 0,Y 377.514,Z 541.099,A -85,B 0,C 180,E1 -12360.649,E2 -12360.649} C_VEL
LIN {X 0,Y 378.412,Z 531.051,A -85,B 0,C 180,E1 -12363.861,E2 -12363.861} C_VEL
LIN {X 0,Y 379.39,Z 522.285,A -85,B 0,C 180,E1 -12366.785,E2 -12366.785} C_VEL
LIN {X 0,Y 379.22,Z 518.228,A -85,B 0,C 180,E1 -12368.249,E2 -12368.249} C_VEL
LIN {X 0,Y 377.837,Z 510.69,A -85,B 0,C 180,E1 -12371.224,E2 -12371.224} C_VEL
LIN {X 0,Y 376.173,Z 502.593,A -85,B 0,C 180,E1 -12374.769,E2 -12374.769} C_VEL
LIN {X 0,Y 375.983,Z 501.657,A -85,B 0,C 180,E1 -12375.26,E2 -12375.26} C_VEL
LIN {X 0,Y 375.942,Z 501.661,A -85,B 0,C 180,E1 -12379.133,E2 -12379.133} C_VEL
LIN {X 0,Y 375.966,Z 501.652,A -85,B 0,C 180,E1 -12381.912,E2 -12381.912} C_VEL
LIN {X 0,Y 375.982,Z 501.651,A -85,B 0,C 180,E1 -12385.333,E2 -12385.333} C_VEL
LIN {X 0,Y 375.96,Z 501.65,A -85,B 0,C 180,E1 -12388.438,E2 -12388.438} C_VEL
LIN {X 0,Y 375.999,Z 501.649,A -85,B 0,C 180,E1 -12392.142,E2 -12392.142} C_VEL
LIN {X 0,Y 376.009,Z 501.647,A -85,B 0,C 180,E1 -12394.539,E2 -12394.539} C_VEL
LIN {X 0,Y 375.966,Z 501.652,A -85,B 0,C 180,E1 -12398.046,E2 -12398.046} C_VEL
LIN {X 0,Y 376.012,Z 501.645,A -85,B 0,C 180,E1 -12401.474,E2 -12401.474} C_VEL
LIN {X 0,Y 376.062,Z 501.638,A -85,B 0,C 180,E1 -12404.833,E2 -12404.833} C_VEL
LIN {X 0,Y 376.053,Z 501.64,A -85,B 0,C 180,E1 -12408.137,E2 -12408.137} C_VEL
LIN {X 0,Y 376.262,Z 501.611,A -85,B 0,C 180,E1 -12411.877,E2 -12411.877} C_VEL
LIN {X 0,Y 376.172,Z 501.625,A -85,B 0,C 180,E1 -12414.64,E2 -12414.64} C_VEL
LIN {X 0,Y 376.348,Z 501.605,A -85,B 0,C 180,E1 -12417.86,E2 -12417.86} C_VEL
LIN {X 0,Y 376.489,Z 501.588,A -85,B 0,C 180,E1 -12420,E2 -12420} C_VEL
LIN {X 0,Y 376.187,Z 501.629,A -85,B 0,C 180,E1 -12423.213,E2 -12423.213} C_VEL
LIN {X 0,Y 376.2,Z 501.62,A -85,B 0,C 180,E1 -12426.49,E2 -12426.49} C_VEL
LIN {X 0,Y 376.123,Z 501.635,A -85,B 0,C 180,E1 -12429.682,E2 -12429.682} C_VEL
LIN {X 0,Y 376.093,Z 501.638,A -85,B 0,C 180,E1 -12433.657,E2 -12433.657} C_VEL
LIN {X 0,Y 376.093,Z 501.646,A -85,B 0,C 180,E1 -12435.097,E2 -12435.097} C_VEL
LIN {X 0,Y 380.008,Z 512.773,A -85,B 0,C 180,E1 -12436.106,E2 -12436.106} C_VEL
LIN {X 0,Y 382.807,Z 522.211,A -85,B 0,C 180,E1 -12437.083,E2 -12437.083} C_VEL
LIN {X 0,Y 381.978,Z 533.762,A -85,B 0,C 180,E1 -12438.227,E2 -12438.227} C_VEL
LIN {X 0,Y 381.108,Z 543.196,A -85,B 0,C 180,E1 -12439.387,E2 -12439.387} C_VEL
LIN {X 0,Y 380.297,Z 551.032,A -85,B 0,C 180,E1 -12440.557,E2 -12440.557} C_VEL
LIN {X 0,Y 379.286,Z 559.526,A -85,B 0,C 180,E1 -12442.107,E2 -12442.107} C_VEL
LIN {X 0,Y 378.407,Z 566.995,A -85,B 0,C 180,E1 -12443.826,E2 -12443.826} C_VEL
LIN {X 0,Y 377.756,Z 572.197,A -85,B 0,C 180,E1 -12445.335,E2 -12445.335} C_VEL
LIN {X 0,Y 377.111,Z 577.109,A -85,B 0,C 180,E1 -12447.167,E2 -12447.167} C_VEL
LIN {X 0,Y 376.604,Z 580.643,A -85,B 0,C 180,E1 -12449.026,E2 -12449.026} C_VEL
LIN {X 0,Y 376.259,Z 582.792,A -85,B 0,C 180,E1 -12450.77,E2 -12450.77} C_VEL
LIN {X 0,Y 375.994,Z 583.964,A -85,B 0,C 180,E1 -12452.825,E2 -12452.825} C_VEL
LIN {X 0,Y 375.908,Z 583.783,A -85,B 0,C 180,E1 -12454.651,E2 -12454.651} C_VEL
LIN {X 0,Y 375.971,Z 582.132,A -85,B 0,C 180,E1 -12456.74,E2 -12456.74} C_VEL
LIN {X 0,Y 376.159,Z 579.018,A -85,B 0,C 180,E1 -12458.808,E2 -12458.808} C_VEL
LIN {X 0,Y 376.582,Z 574.463,A -85,B 0,C 180,E1 -12460.783,E2 -12460.783} C_VEL
LIN {X 0,Y 377.023,Z 569.247,A -85,B 0,C 180,E1 -12462.477,E2 -12462.477} C_VEL
LIN {X 0,Y 377.642,Z 562.252,A -85,B 0,C 180,E1 -12464.258,E2 -12464.258} C_VEL
LIN {X 0,Y 378.271,Z 555.35,A -85,B 0,C 180,E1 -12465.668,E2 -12465.668} C_VEL
LIN {X 0,Y 379.029,Z 546.284,A -85,B 0,C 180,E1 -12467.178,E2 -12467.178} C_VEL
LIN {X 0,Y 379.811,Z 536.416,A -85,B 0,C 180,E1 -12468.515,E2 -12468.515} C_VEL
LIN {X 0,Y 380.547,Z 525.283,A -85,B 0,C 180,E1 -12469.73,E2 -12469.73} C_VEL
LIN {X 0,Y 380.897,Z 519.121,A -85,B 0,C 180,E1 -12470.292,E2 -12470.292} C_VEL
LIN {X 0,Y 377.615,Z 507.244,A -85,B 0,C 180,E1 -12471.384,E2 -12471.384} C_VEL
LIN {X 0,Y 375.966,Z 501.655,A -85,B 0,C 180,E1 -12471.844,E2 -12471.844} C_VEL
LIN {X 0,Y 375.985,Z 501.653,A -85,B 0,C 180,E1 -12475.333,E2 -12475.333} C_VEL
LIN {X 0,Y 375.963,Z 501.652,A -85,B 0,C 180,E1 -12478.438,E2 -12478.438} C_VEL
LIN {X 0,Y 376.001,Z 501.647,A -85,B 0,C 180,E1 -12482.141,E2 -12482.141} C_VEL
LIN {X 0,Y 376.009,Z 501.646,A -85,B 0,C 180,E1 -12484.539,E2 -12484.539} C_VEL
LIN {X 0,Y 375.962,Z 501.652,A -85,B 0,C 180,E1 -12488.045,E2 -12488.045} C_VEL
LIN {X 0,Y 376.008,Z 501.65,A -85,B 0,C 180,E1 -12491.473,E2 -12491.473} C_VEL
LIN {X 0,Y 376.063,Z 501.64,A -85,B 0,C 180,E1 -12494.833,E2 -12494.833} C_VEL
LIN {X 0,Y 376.055,Z 501.64,A -85,B 0,C 180,E1 -12498.137,E2 -12498.137} C_VEL
LIN {X 0,Y 376.192,Z 501.624,A -85,B 0,C 180,E1 -12501.953,E2 -12501.953} C_VEL
LIN {X 0,Y 376.16,Z 501.627,A -85,B 0,C 180,E1 -12504.64,E2 -12504.64} C_VEL
LIN {X 0,Y 376.357,Z 501.604,A -85,B 0,C 180,E1 -12507.859,E2 -12507.859} C_VEL
LIN {X 0,Y 376.464,Z 501.589,A -85,B 0,C 180,E1 -12510,E2 -12510} C_VEL
LIN {X 0,Y 376.355,Z 501.602,A -85,B 0,C 180,E1 -12512.14,E2 -12512.14} C_VEL
LIN {X 0,Y 376.205,Z 501.621,A -85,B 0,C 180,E1 -12516.436,E2 -12516.436} C_VEL
LIN {X 0,Y 376.118,Z 501.634,A -85,B 0,C 180,E1 -12519.681,E2 -12519.681} C_VEL
LIN {X 0,Y 376.094,Z 501.637,A -85,B 0,C 180,E1 -12523.657,E2 -12523.657} C_VEL
LIN {X 0,Y 376.037,Z 501.647,A -85,B 0,C 180,E1 -12527.4,E2 -12527.4} C_VEL
LIN {X 0,Y 375.983,Z 501.651,A -85,B 0,C 180,E1 -12530.832,E2 -12530.832} C_VEL
LIN {X 0,Y 375.987,Z 501.648,A -85,B 0,C 180,E1 -12534.282,E2 -12534.282} C_VEL
LIN {X 0,Y 375.968,Z 501.652,A -85,B 0,C 180,E1 -12536.656,E2 -12536.656} C_VEL
LIN {X 0,Y 375.967,Z 501.651,A -85,B 0,C 180,E1 -12540.312,E2 -12540.312} C_VEL
LIN {X 0,Y 375.934,Z 501.654,A -85,B 0,C 180,E1 -12543.371,E2 -12543.371} C_VEL
LIN {X 0,Y 375.272,Z 501.738,A -85,B 0,C 180,E1 -12544.266,E2 -12544.266} C_VEL
LIN {X 0,Y 372.421,Z 502.094,A -85,B 0,C 180,E1 -12545.72,E2 -12545.72} C_VEL
LIN {X 0,Y 370.002,Z 502.397,A -85,B 0,C 180,E1 -12546.897,E2 -12546.897} C_VEL
LIN {X 0,Y 368.961,Z 502.524,A -85,B 0,C 180,E1 -12547.806,E2 -12547.806} C_VEL
LIN {X 0,Y 368.874,Z 502.534,A -85,B 0,C 180,E1 -12548.115,E2 -12548.115} C_VEL
LIN {X 0,Y 368.872,Z 502.535,A -85,B 0,C 180,E1 -12551.824,E2 -12551.824} C_VEL
LIN {X 0,Y 368.882,Z 502.537,A -85,B 0,C 180,E1 -12555.175,E2 -12555.175} C_VEL
LIN {X 0,Y 368.884,Z 502.533,A -85,B 0,C 180,E1 -12558.177,E2 -12558.177} C_VEL
LIN {X 0,Y 368.908,Z 502.534,A -85,B 0,C 180,E1 -12561.36,E2 -12561.36} C_VEL
LIN {X 0,Y 368.939,Z 502.531,A -85,B 0,C 180,E1 -12565.146,E2 -12565.146} C_VEL
LIN {X 0,Y 368.932,Z 502.531,A -85,B 0,C 180,E1 -12569.046,E2 -12569.046} C_VEL
LIN {X 0,Y 368.979,Z 502.522,A -85,B 0,C 180,E1 -12571.563,E2 -12571.563} C_VEL
LIN {X 0,Y 369.002,Z 502.518,A -85,B 0,C 180,E1 -12574.019,E2 -12574.019} C_VEL
LIN {X 0,Y 368.925,Z 502.528,A -85,B 0,C 180,E1 -12577.604,E2 -12577.604} C_VEL
LIN {X 0,Y 368.96,Z 502.528,A -85,B 0,C 180,E1 -12581.106,E2 -12581.106} C_VEL
LIN {X 0,Y 369,Z 502.52,A -85,B 0,C 180,E1 -12584.535,E2 -12584.535} C_VEL
LIN {X 0,Y 369.007,Z 502.518,A -85,B 0,C 180,E1 -12587.906,E2 -12587.906} C_VEL
LIN {X 0,Y 369.093,Z 502.51,A -85,B 0,C 180,E1 -12591.238,E2 -12591.238} C_VEL
LIN {X 0,Y 369.133,Z 502.504,A -85,B 0,C 180,E1 -12594.537,E2 -12594.537} C_VEL
LIN {X 0,Y 369.316,Z 502.479,A -85,B 0,C 180,E1 -12597.819,E2 -12597.819} C_VEL
LIN {X 0,Y 369.455,Z 502.462,A -85,B 0,C 180,E1 -12600,E2 -12600} C_VEL
LIN {X 0,Y 369.309,Z 502.48,A -85,B 0,C 180,E1 -12602.181,E2 -12602.181} C_VEL
LIN {X 0,Y 369.163,Z 502.501,A -85,B 0,C 180,E1 -12606.559,E2 -12606.559} C_VEL
LIN {X 0,Y 369.071,Z 502.51,A -85,B 0,C 180,E1 -12609.868,E2 -12609.868} C_VEL
LIN {X 0,Y 369.039,Z 502.513,A -85,B 0,C 180,E1 -12613.772,E2 -12613.772} C_VEL
LIN {X 0,Y 368.992,Z 502.52,A -85,B 0,C 180,E1 -12617.743,E2 -12617.743} C_VEL
LIN {X 0,Y 368.911,Z 502.532,A -85,B 0,C 180,E1 -12621.221,E2 -12621.221} C_VEL
LIN {X 0,Y 368.937,Z 502.531,A -85,B 0,C 180,E1 -12624.777,E2 -12624.777} C_VEL
LIN {X 0,Y 368.917,Z 502.532,A -85,B 0,C 180,E1 -12628.441,E2 -12628.441} C_VEL
LIN {X 0,Y 368.911,Z 502.533,A -85,B 0,C 180,E1 -12630.987,E2 -12630.987} C_VEL
LIN {X 0,Y 368.937,Z 502.531,A -85,B 0,C 180,E1 -12634.853,E2 -12634.853} C_VEL
LIN {X 0,Y 368.907,Z 502.535,A -85,B 0,C 180,E1 -12638.64,E2 -12638.64} C_VEL
LIN {X 0,Y 368.882,Z 502.536,A -85,B 0,C 180,E1 -12642.009,E2 -12642.009} C_VEL
LIN {X 0,Y 368.916,Z 502.54,A -85,B 0,C 180,E1 -12644.492,E2 -12644.492} C_VEL
LIN {X 0,Y 370.549,Z 510.834,A -85,B 0,C 180,E1 -12647.705,E2 -12647.705} C_VEL
LIN {X 0,Y 372.58,Z 521.144,A -85,B 0,C 180,E1 -12651.502,E2 -12651.502} C_VEL
LIN {X 0,Y 372.973,Z 523.441,A -85,B 0,C 180,E1 -12652.318,E2 -12652.318} C_VEL
LIN {X 0,Y 372.294,Z 531.122,A -85,B 0,C 180,E1 -12654.854,E2 -12654.854} C_VEL
LIN {X 0,Y 371.13,Z 543.509,A -85,B 0,C 180,E1 -12658.831,E2 -12658.831} C_VEL
LIN {X 0,Y 369.872,Z 557.665,A -85,B 0,C 180,E1 -12663.26,E2 -12663.26} C_VEL
LIN {X 0,Y 369.067,Z 569.901,A -85,B 0,C 180,E1 -12667.022,E2 -12667.022} C_VEL
LIN {X 0,Y 368.481,Z 581.988,A -85,B 0,C 180,E1 -12670.683,E2 -12670.683} C_VEL
LIN {X 0,Y 370.255,Z 598.893,A -85,B 0,C 180,E1 -12671.383,E2 -12671.383} C_VEL
LIN {X 0,Y 371.134,Z 612.069,A -85,B 0,C 180,E1 -12672.144,E2 -12672.144} C_VEL
LIN {X 0,Y 371.625,Z 624.758,A -85,B 0,C 180,E1 -12673.096,E2 -12673.096} C_VEL
LIN {X 0,Y 371.412,Z 632.399,A -85,B 0,C 180,E1 -12673.793,E2 -12673.793} C_VEL
LIN {X 0,Y 370.481,Z 642.558,A -85,B 0,C 180,E1 -12674.88,E2 -12674.88} C_VEL
LIN {X 0,Y 369.544,Z 651.603,A -85,B 0,C 180,E1 -12676.06,E2 -12676.06} C_VEL
LIN {X 0,Y 369.165,Z 658.142,A -85,B 0,C 180,E1 -12677.074,E2 -12677.074} C_VEL
LIN {X 0,Y 368.518,Z 667.066,A -85,B 0,C 180,E1 -12678.727,E2 -12678.727} C_VEL
LIN {X 0,Y 368.196,Z 674.239,A -85,B 0,C 180,E1 -12680.386,E2 -12680.386} C_VEL
LIN {X 0,Y 368.061,Z 680.775,A -85,B 0,C 180,E1 -12682.319,E2 -12682.319} C_VEL
LIN {X 0,Y 368.109,Z 685.061,A -85,B 0,C 180,E1 -12683.973,E2 -12683.973} C_VEL
LIN {X 0,Y 368.368,Z 688.25,A -85,B 0,C 180,E1 -12685.623,E2 -12685.623} C_VEL
LIN {X 0,Y 368.36,Z 689.782,A -85,B 0,C 180,E1 -12686.719,E2 -12686.719} C_VEL
LIN {X 0,Y 368.401,Z 690.866,A -85,B 0,C 180,E1 -12687.814,E2 -12687.814} C_VEL
LIN {X 0,Y 368.698,Z 691.742,A -85,B 0,C 180,E1 -12690,E2 -12690} C_VEL
LIN {X 0,Y 368.464,Z 691.505,A -85,B 0,C 180,E1 -12691.093,E2 -12691.093} C_VEL
LIN {X 0,Y 368.397,Z 690.85,A -85,B 0,C 180,E1 -12692.187,E2 -12692.187} C_VEL
LIN {X 0,Y 368.351,Z 689.753,A -85,B 0,C 180,E1 -12693.282,E2 -12693.282} C_VEL
LIN {X 0,Y 368.318,Z 688.241,A -85,B 0,C 180,E1 -12694.378,E2 -12694.378} C_VEL
LIN {X 0,Y 368.122,Z 685.101,A -85,B 0,C 180,E1 -12696.028,E2 -12696.028} C_VEL
LIN {X 0,Y 368.065,Z 680.902,A -85,B 0,C 180,E1 -12697.681,E2 -12697.681} C_VEL
LIN {X 0,Y 368.147,Z 674.55,A -85,B 0,C 180,E1 -12699.616,E2 -12699.616} C_VEL
LIN {X 0,Y 368.491,Z 667.648,A -85,B 0,C 180,E1 -12701.274,E2 -12701.274} C_VEL
LIN {X 0,Y 369.143,Z 659.158,A -85,B 0,C 180,E1 -12702.927,E2 -12702.927} C_VEL
LIN {X 0,Y 369.807,Z 650.589,A -85,B 0,C 180,E1 -12704.304,E2 -12704.304} C_VEL
LIN {X 0,Y 370.85,Z 640.315,A -85,B 0,C 180,E1 -12705.668,E2 -12705.668} C_VEL
LIN {X 0,Y 372.109,Z 628.906,A -85,B 0,C 180,E1 -12706.881,E2 -12706.881} C_VEL
LIN {X 0,Y 371.993,Z 616.482,A -85,B 0,C 180,E1 -12707.991,E2 -12707.991} C_VEL
LIN {X 0,Y 371.769,Z 604.835,A -85,B 0,C 180,E1 -12708.825,E2 -12708.825} C_VEL
LIN {X 0,Y 370.743,Z 591.497,A -85,B 0,C 180,E1 -12709.59,E2 -12709.59} C_VEL
LIN {X 0,Y 368.521,Z 576.176,A -85,B 0,C 180,E1 -12710.309,E2 -12710.309} C_VEL
LIN {X 0,Y 369.092,Z 562.843,A -85,B 0,C 180,E1 -12714.277,E2 -12714.277} C_VEL
LIN {X 0,Y 369.801,Z 551.478,A -85,B 0,C 180,E1 -12717.751,E2 -12717.751} C_VEL
LIN {X 0,Y 370.656,Z 539.853,A -85,B 0,C 180,E1 -12721.434,E2 -12721.434} C_VEL
LIN {X 0,Y 371.624,Z 530.353,A -85,B 0,C 180,E1 -12724.566,E2 -12724.566} C_VEL
LIN {X 0,Y 372.489,Z 522.871,A -85,B 0,C 180,E1 -12727.14,E2 -12727.14} C_VEL
LIN {X 0,Y 372.177,Z 519.126,A -85,B 0,C 180,E1 -12728.547,E2 -12728.547} C_VEL
LIN {X 0,Y 370.836,Z 511.727,A -85,B 0,C 180,E1 -12731.553,E2 -12731.553} C_VEL
LIN {X 0,Y 369.179,Z 503.63,A -85,B 0,C 180,E1 -12735.222,E2 -12735.222} C_VEL
LIN {X 0,Y 368.901,Z 502.54,A -85,B 0,C 180,E1 -12735.831,E2 -12735.831} C_VEL
LIN {X 0,Y 368.914,Z 502.534,A -85,B 0,C 180,E1 -12739.643,E2 -12739.643} C_VEL
LIN {X 0,Y 368.903,Z 502.534,A -85,B 0,C 180,E1 -12743.145,E2 -12743.145} C_VEL
LIN {X 0,Y 368.899,Z 502.533,A -85,B 0,C 180,E1 -12746.462,E2 -12746.462} C_VEL
LIN {X 0,Y 368.932,Z 502.53,A -85,B 0,C 180,E1 -12749.047,E2 -12749.047} C_VEL
LIN {X 0,Y 368.983,Z 502.522,A -85,B 0,C 180,E1 -12751.564,E2 -12751.564} C_VEL
LIN {X 0,Y 369.003,Z 502.518,A -85,B 0,C 180,E1 -12754.02,E2 -12754.02} C_VEL
LIN {X 0,Y 368.935,Z 502.529,A -85,B 0,C 180,E1 -12757.605,E2 -12757.605} C_VEL
LIN {X 0,Y 368.961,Z 502.525,A -85,B 0,C 180,E1 -12761.106,E2 -12761.106} C_VEL
LIN {X 0,Y 369.001,Z 502.52,A -85,B 0,C 180,E1 -12764.536,E2 -12764.536} C_VEL
LIN {X 0,Y 369.008,Z 502.519,A -85,B 0,C 180,E1 -12767.907,E2 -12767.907} C_VEL
LIN {X 0,Y 369.233,Z 502.487,A -85,B 0,C 180,E1 -12771.801,E2 -12771.801} C_VEL
LIN {X 0,Y 369.145,Z 502.501,A -85,B 0,C 180,E1 -12774.538,E2 -12774.538} C_VEL
LIN {X 0,Y 369.312,Z 502.481,A -85,B 0,C 180,E1 -12777.819,E2 -12777.819} C_VEL
LIN {X 0,Y 369.459,Z 502.464,A -85,B 0,C 180,E1 -12780,E2 -12780} C_VEL
LIN {X 0,Y 369.32,Z 502.482,A -85,B 0,C 180,E1 -12782.181,E2 -12782.181} C_VEL
LIN {X 0,Y 369.166,Z 502.497,A -85,B 0,C 180,E1 -12786.559,E2 -12786.559} C_VEL
LIN {X 0,Y 369.071,Z 502.515,A -85,B 0,C 180,E1 -12789.869,E2 -12789.869} C_VEL
LIN {X 0,Y 369.04,Z 502.517,A -85,B 0,C 180,E1 -12793.772,E2 -12793.772} C_VEL
LIN {X 0,Y 369.038,Z 502.517,A -85,B 0,C 180,E1 -12794.616,E2 -12794.616} C_VEL
LIN {X 0,Y 373.219,Z 514.059,A -85,B 0,C 180,E1 -12795.706,E2 -12795.706} C_VEL
LIN {X 0,Y 376.176,Z 524.147,A -85,B 0,C 180,E1 -12796.795,E2 -12796.795} C_VEL
LIN {X 0,Y 375.298,Z 535.365,A -85,B 0,C 180,E1 -12797.942,E2 -12797.942} C_VEL
LIN {X 0,Y 374.325,Z 545.135,A -85,B 0,C 180,E1 -12799.182,E2 -12799.182} C_VEL
LIN {X 0,Y 373.257,Z 554.558,A -85,B 0,C 180,E1 -12800.674,E2 -12800.674} C_VEL
LIN {X 0,Y 372.256,Z 562.885,A -85,B 0,C 180,E1 -12802.316,E2 -12802.316} C_VEL
LIN {X 0,Y 371.349,Z 569.659,A -85,B 0,C 180,E1 -12804.011,E2 -12804.011} C_VEL
LIN {X 0,Y 370.549,Z 575.419,A -85,B 0,C 180,E1 -12805.864,E2 -12805.864} C_VEL
LIN {X 0,Y 369.973,Z 579.751,A -85,B 0,C 180,E1 -12807.737,E2 -12807.737} C_VEL
LIN {X 0,Y 369.458,Z 582.77,A -85,B 0,C 180,E1 -12809.643,E2 -12809.643} C_VEL
LIN {X 0,Y 369.21,Z 584.201,A -85,B 0,C 180,E1 -12811.064,E2 -12811.064} C_VEL
LIN {X 0,Y 368.978,Z 585.054,A -85,B 0,C 180,E1 -12813.062,E2 -12813.062} C_VEL
LIN {X 0,Y 368.902,Z 584.616,A -85,B 0,C 180,E1 -12814.995,E2 -12814.995} C_VEL
LIN {X 0,Y 368.947,Z 583.021,A -85,B 0,C 180,E1 -12816.865,E2 -12816.865} C_VEL
LIN {X 0,Y 369.176,Z 579.904,A -85,B 0,C 180,E1 -12818.92,E2 -12818.92} C_VEL
LIN {X 0,Y 369.634,Z 575.027,A -85,B 0,C 180,E1 -12821.024,E2 -12821.024} C_VEL
LIN {X 0,Y 370.04,Z 570.197,A -85,B 0,C 180,E1 -12822.6,E2 -12822.6} C_VEL
LIN {X 0,Y 370.539,Z 564.419,A -85,B 0,C 180,E1 -12824.12,E2 -12824.12} C_VEL
LIN {X 0,Y 371.277,Z 557.012,A -85,B 0,C 180,E1 -12825.702,E2 -12825.702} C_VEL
LIN {X 0,Y 371.972,Z 548.78,A -85,B 0,C 180,E1 -12827.142,E2 -12827.142} C_VEL
LIN {X 0,Y 372.846,Z 538.206,A -85,B 0,C 180,E1 -12828.63,E2 -12828.63} C_VEL
LIN {X 0,Y 373.615,Z 527.607,A -85,B 0,C 180,E1 -12829.836,E2 -12829.836} C_VEL
LIN {X 0,Y 374.001,Z 521.756,A -85,B 0,C 180,E1 -12830.395,E2 -12830.395} C_VEL
LIN {X 0,Y 373.387,Z 518.014,A -85,B 0,C 180,E1 -12830.763,E2 -12830.763} C_VEL
LIN {X 0,Y 370.309,Z 507.312,A -85,B 0,C 180,E1 -12831.743,E2 -12831.743} C_VEL
LIN {X 0,Y 368.928,Z 502.532,A -85,B 0,C 180,E1 -12832.138,E2 -12832.138} C_VEL
LIN {X 0,Y 368.941,Z 502.529,A -85,B 0,C 180,E1 -12835.147,E2 -12835.147} C_VEL
LIN {X 0,Y 368.934,Z 502.53,A -85,B 0,C 180,E1 -12839.047,E2 -12839.047} C_VEL
LIN {X 0,Y 368.985,Z 502.524,A -85,B 0,C 180,E1 -12841.564,E2 -12841.564} C_VEL
LIN {X 0,Y 369.004,Z 502.519,A -85,B 0,C 180,E1 -12844.02,E2 -12844.02} C_VEL
LIN {X 0,Y 368.927,Z 502.531,A -85,B 0,C 180,E1 -12847.604,E2 -12847.604} C_VEL
LIN {X 0,Y 368.959,Z 502.528,A -85,B 0,C 180,E1 -12851.106,E2 -12851.106} C_VEL
LIN {X 0,Y 369.002,Z 502.518,A -85,B 0,C 180,E1 -12854.535,E2 -12854.535} C_VEL
LIN {X 0,Y 369.01,Z 502.518,A -85,B 0,C 180,E1 -12857.907,E2 -12857.907} C_VEL
LIN {X 0,Y 369.096,Z 502.511,A -85,B 0,C 180,E1 -12861.238,E2 -12861.238} C_VEL
LIN {X 0,Y 369.131,Z 502.502,A -85,B 0,C 180,E1 -12864.537,E2 -12864.537} C_VEL
LIN {X 0,Y 369.322,Z 502.48,A -85,B 0,C 180,E1 -12867.819,E2 -12867.819} C_VEL
LIN {X 0,Y 369.414,Z 502.467,A -85,B 0,C 180,E1 -12870,E2 -12870} C_VEL
LIN {X 0,Y 369.319,Z 502.478,A -85,B 0,C 180,E1 -12872.181,E2 -12872.181} C_VEL
LIN {X 0,Y 369.166,Z 502.498,A -85,B 0,C 180,E1 -12876.559,E2 -12876.559} C_VEL
LIN {X 0,Y 369.068,Z 502.511,A -85,B 0,C 180,E1 -12879.868,E2 -12879.868} C_VEL
LIN {X 0,Y 369.042,Z 502.514,A -85,B 0,C 180,E1 -12883.772,E2 -12883.772} C_VEL
LIN {X 0,Y 368.995,Z 502.521,A -85,B 0,C 180,E1 -12887.743,E2 -12887.743} C_VEL
LIN {X 0,Y 368.933,Z 502.531,A -85,B 0,C 180,E1 -12891.219,E2 -12891.219} C_VEL
LIN {X 0,Y 368.945,Z 502.528,A -85,B 0,C 180,E1 -12894.776,E2 -12894.776} C_VEL
LIN {X 0,Y 368.934,Z 502.527,A -85,B 0,C 180,E1 -12898.44,E2 -12898.44} C_VEL
LIN {X 0,Y 368.914,Z 502.533,A -85,B 0,C 180,E1 -12900.987,E2 -12900.987} C_VEL
LIN {X 0,Y 368.94,Z 502.53,A -85,B 0,C 180,E1 -12904.853,E2 -12904.853} C_VEL
LIN {X 0,Y 368.874,Z 502.534,A -85,B 0,C 180,E1 -12908.115,E2 -12908.115} C_VEL
LIN {X 0,Y 368.213,Z 502.622,A -85,B 0,C 180,E1 -12909.026,E2 -12909.026} C_VEL
LIN {X 0,Y 365.391,Z 502.976,A -85,B 0,C 180,E1 -12910.509,E2 -12910.509} C_VEL
LIN {X 0,Y 362.984,Z 503.277,A -85,B 0,C 180,E1 -12911.708,E2 -12911.708} C_VEL
LIN {X 0,Y 361.927,Z 503.404,A -85,B 0,C 180,E1 -12912.635,E2 -12912.635} C_VEL
LIN {X 0,Y 361.827,Z 503.414,A -85,B 0,C 180,E1 -12912.95,E2 -12912.95} C_VEL
LIN {X 0,Y 361.82,Z 503.413,A -85,B 0,C 180,E1 -12915.946,E2 -12915.946} C_VEL
LIN {X 0,Y 361.837,Z 503.415,A -85,B 0,C 180,E1 -12919.245,E2 -12919.245} C_VEL
LIN {X 0,Y 361.865,Z 503.411,A -85,B 0,C 180,E1 -12922.777,E2 -12922.777} C_VEL
LIN {X 0,Y 361.857,Z 503.408,A -85,B 0,C 180,E1 -12925.719,E2 -12925.719} C_VEL
LIN {X 0,Y 361.877,Z 503.406,A -85,B 0,C 180,E1 -12929.672,E2 -12929.672} C_VEL
LIN {X 0,Y 361.956,Z 503.398,A -85,B 0,C 180,E1 -12933.475,E2 -12933.475} C_VEL
LIN {X 0,Y 361.882,Z 503.409,A -85,B 0,C 180,E1 -12937.144,E2 -12937.144} C_VEL
LIN {X 0,Y 361.909,Z 503.405,A -85,B 0,C 180,E1 -12940.723,E2 -12940.723} C_VEL
LIN {X 0,Y 361.935,Z 503.403,A -85,B 0,C 180,E1 -12943.066,E2 -12943.066} C_VEL
LIN {X 0,Y 362.001,Z 503.392,A -85,B 0,C 180,E1 -12946.528,E2 -12946.528} C_VEL
LIN {X 0,Y 362.003,Z 503.389,A -85,B 0,C 180,E1 -12949.937,E2 -12949.937} C_VEL
LIN {X 0,Y 362.137,Z 503.376,A -85,B 0,C 180,E1 -12953.313,E2 -12953.313} C_VEL
LIN {X 0,Y 362.28,Z 503.356,A -85,B 0,C 180,E1 -12957.776,E2 -12957.776} C_VEL
LIN {X 0,Y 362.404,Z 503.34,A -85,B 0,C 180,E1 -12960,E2 -12960} C_VEL
LIN {X 0,Y 362.272,Z 503.357,A -85,B 0,C 180,E1 -12962.223,E2 -12962.223} C_VEL
LIN {X 0,Y 362.126,Z 503.378,A -85,B 0,C 180,E1 -12966.687,E2 -12966.687} C_VEL
LIN {X 0,Y 362.035,Z 503.386,A -85,B 0,C 180,E1 -12970.062,E2 -12970.062} C_VEL
LIN {X 0,Y 362,Z 503.39,A -85,B 0,C 180,E1 -12973.899,E2 -12973.899} C_VEL
LIN {X 0,Y 361.93,Z 503.404,A -85,B 0,C 180,E1 -12976.934,E2 -12976.934} C_VEL
LIN {X 0,Y 361.888,Z 503.406,A -85,B 0,C 180,E1 -12980.461,E2 -12980.461} C_VEL
LIN {X 0,Y 361.894,Z 503.404,A -85,B 0,C 180,E1 -12984.113,E2 -12984.113} C_VEL
LIN {X 0,Y 361.849,Z 503.409,A -85,B 0,C 180,E1 -12987.784,E2 -12987.784} C_VEL
LIN {X 0,Y 361.847,Z 503.41,A -85,B 0,C 180,E1 -12991.285,E2 -12991.285} C_VEL
LIN {X 0,Y 361.855,Z 503.41,A -85,B 0,C 180,E1 -12994.28,E2 -12994.28} C_VEL
LIN {X 0,Y 361.863,Z 503.409,A -85,B 0,C 180,E1 -12997.223,E2 -12997.223} C_VEL
LIN {X 0,Y 361.836,Z 503.415,A -85,B 0,C 180,E1 -13000.755,E2 -13000.755} C_VEL
LIN {X 0,Y 361.88,Z 503.463,A -85,B 0,C 180,E1 -13004.161,E2 -13004.161} C_VEL
LIN {X 0,Y 363.504,Z 511.673,A -85,B 0,C 180,E1 -13007.414,E2 -13007.414} C_VEL
LIN {X 0,Y 365.322,Z 521.053,A -85,B 0,C 180,E1 -13010.947,E2 -13010.947} C_VEL
LIN {X 0,Y 365.974,Z 525.166,A -85,B 0,C 180,E1 -13012.431,E2 -13012.431} C_VEL
LIN {X 0,Y 365.287,Z 532.037,A -85,B 0,C 180,E1 -13014.747,E2 -13014.747} C_VEL
LIN {X 0,Y 364.142,Z 543.763,A -85,B 0,C 180,E1 -13018.594,E2 -13018.594} C_VEL
LIN {X 0,Y 362.844,Z 557.507,A -85,B 0,C 180,E1 -13022.997,E2 -13022.997} C_VEL
LIN {X 0,Y 362.073,Z 568.803,A -85,B 0,C 180,E1 -13026.552,E2 -13026.552} C_VEL
LIN {X 0,Y 361.463,Z 581.102,A -85,B 0,C 180,E1 -13030.366,E2 -13030.366} C_VEL
LIN {X 0,Y 363.127,Z 597.321,A -85,B 0,C 180,E1 -13031.04,E2 -13031.04} C_VEL
LIN {X 0,Y 363.975,Z 609.749,A -85,B 0,C 180,E1 -13031.76,E2 -13031.76} C_VEL
LIN {X 0,Y 364.475,Z 621.2,A -85,B 0,C 180,E1 -13032.61,E2 -13032.61} C_VEL
LIN {X 0,Y 364.563,Z 630.817,A -85,B 0,C 180,E1 -13033.48,E2 -13033.48} C_VEL
LIN {X 0,Y 363.544,Z 641.067,A -85,B 0,C 180,E1 -13034.585,E2 -13034.585} C_VEL
LIN {X 0,Y 362.492,Z 651.283,A -85,B 0,C 180,E1 -13035.942,E2 -13035.942} C_VEL
LIN {X 0,Y 361.873,Z 660.026,A -85,B 0,C 180,E1 -13037.38,E2 -13037.38} C_VEL
LIN {X 0,Y 361.331,Z 668.359,A -85,B 0,C 180,E1 -13039.068,E2 -13039.068} C_VEL
LIN {X 0,Y 361.07,Z 675.082,A -85,B 0,C 180,E1 -13040.759,E2 -13040.759} C_VEL
LIN {X 0,Y 361,Z 679.61,A -85,B 0,C 180,E1 -13042.168,E2 -13042.168} C_VEL
LIN {X 0,Y 361.044,Z 683.931,A -85,B 0,C 180,E1 -13043.854,E2 -13043.854} C_VEL
LIN {X 0,Y 361.311,Z 687.152,A -85,B 0,C 180,E1 -13045.538,E2 -13045.538} C_VEL
LIN {X 0,Y 361.323,Z 688.699,A -85,B 0,C 180,E1 -13046.655,E2 -13046.655} C_VEL
LIN {X 0,Y 361.366,Z 689.806,A -85,B 0,C 180,E1 -13047.771,E2 -13047.771} C_VEL
LIN {X 0,Y 361.672,Z 690.704,A -85,B 0,C 180,E1 -13050,E2 -13050} C_VEL
LIN {X 0,Y 361.432,Z 690.474,A -85,B 0,C 180,E1 -13051.114,E2 -13051.114} C_VEL
LIN {X 0,Y 361.355,Z 689.84,A -85,B 0,C 180,E1 -13052.229,E2 -13052.229} C_VEL
LIN {X 0,Y 361.302,Z 688.753,A -85,B 0,C 180,E1 -13053.346,E2 -13053.346} C_VEL
LIN {X 0,Y 361.246,Z 687.245,A -85,B 0,C 180,E1 -13054.463,E2 -13054.463} C_VEL
LIN {X 0,Y 361.06,Z 684.123,A -85,B 0,C 180,E1 -13056.146,E2 -13056.146} C_VEL
LIN {X 0,Y 360.997,Z 679.939,A -85,B 0,C 180,E1 -13057.833,E2 -13057.833} C_VEL
LIN {X 0,Y 361.097,Z 673.608,A -85,B 0,C 180,E1 -13059.805,E2 -13059.805} C_VEL
LIN {X 0,Y 361.484,Z 666.75,A -85,B 0,C 180,E1 -13061.495,E2 -13061.495} C_VEL
LIN {X 0,Y 362.187,Z 658.325,A -85,B 0,C 180,E1 -13063.18,E2 -13063.18} C_VEL
LIN {X 0,Y 362.644,Z 651.688,A -85,B 0,C 180,E1 -13064.305,E2 -13064.305} C_VEL
LIN {X 0,Y 363.775,Z 641.838,A -85,B 0,C 180,E1 -13065.693,E2 -13065.693} C_VEL
LIN {X 0,Y 365.148,Z 629.77,A -85,B 0,C 180,E1 -13067.069,E2 -13067.069} C_VEL
LIN {X 0,Y 365.123,Z 617.825,A -85,B 0,C 180,E1 -13068.198,E2 -13068.198} C_VEL
LIN {X 0,Y 365.004,Z 605.85,A -85,B 0,C 180,E1 -13069.107,E2 -13069.107} C_VEL
LIN {X 0,Y 364.027,Z 592.047,A -85,B 0,C 180,E1 -13069.967,E2 -13069.967} C_VEL
LIN {X 0,Y 362.094,Z 578.382,A -85,B 0,C 180,E1 -13070.637,E2 -13070.637} C_VEL
LIN {X 0,Y 361.494,Z 574.977,A -85,B 0,C 180,E1 -13070.796,E2 -13070.796} C_VEL
LIN {X 0,Y 362.105,Z 562.313,A -85,B 0,C 180,E1 -13074.663,E2 -13074.663} C_VEL
LIN {X 0,Y 362.737,Z 552.589,A -85,B 0,C 180,E1 -13077.71,E2 -13077.71} C_VEL
LIN {X 0,Y 363.743,Z 540.058,A -85,B 0,C 180,E1 -13081.773,E2 -13081.773} C_VEL
LIN {X 0,Y 364.871,Z 529.683,A -85,B 0,C 180,E1 -13085.3,E2 -13085.3} C_VEL
LIN {X 0,Y 365.563,Z 524.13,A -85,B 0,C 180,E1 -13087.268,E2 -13087.268} C_VEL
LIN {X 0,Y 365.2,Z 520.376,A -85,B 0,C 180,E1 -13088.715,E2 -13088.715} C_VEL
LIN {X 0,Y 363.796,Z 512.662,A -85,B 0,C 180,E1 -13091.948,E2 -13091.948} C_VEL
LIN {X 0,Y 362.489,Z 506.182,A -85,B 0,C 180,E1 -13094.954,E2 -13094.954} C_VEL
LIN {X 0,Y 361.866,Z 503.417,A -85,B 0,C 180,E1 -13096.376,E2 -13096.376} C_VEL
LIN {X 0,Y 361.857,Z 503.411,A -85,B 0,C 180,E1 -13100.139,E2 -13100.139} C_VEL
LIN {X 0,Y 361.869,Z 503.411,A -85,B 0,C 180,E1 -13102.982,E2 -13102.982} C_VEL
LIN {X 0,Y 361.861,Z 503.411,A -85,B 0,C 180,E1 -13106.631,E2 -13106.631} C_VEL
LIN {X 0,Y 361.877,Z 503.409,A -85,B 0,C 180,E1 -13109.672,E2 -13109.672} C_VEL
LIN {X 0,Y 361.957,Z 503.392,A -85,B 0,C 180,E1 -13113.475,E2 -13113.475} C_VEL
LIN {X 0,Y 361.893,Z 503.405,A -85,B 0,C 180,E1 -13117.145,E2 -13117.145} C_VEL
LIN {X 0,Y 361.91,Z 503.405,A -85,B 0,C 180,E1 -13120.724,E2 -13120.724} C_VEL
LIN {X 0,Y 361.936,Z 503.4,A -85,B 0,C 180,E1 -13123.066,E2 -13123.066} C_VEL
LIN {X 0,Y 362.002,Z 503.394,A -85,B 0,C 180,E1 -13126.528,E2 -13126.528} C_VEL
LIN {X 0,Y 362.035,Z 503.39,A -85,B 0,C 180,E1 -13129.938,E2 -13129.938} C_VEL
LIN {X 0,Y 362.155,Z 503.369,A -85,B 0,C 180,E1 -13132.193,E2 -13132.193} C_VEL
LIN {X 0,Y 362.119,Z 503.377,A -85,B 0,C 180,E1 -13134.432,E2 -13134.432} C_VEL
LIN {X 0,Y 362.275,Z 503.358,A -85,B 0,C 180,E1 -13137.777,E2 -13137.777} C_VEL
LIN {X 0,Y 362.429,Z 503.34,A -85,B 0,C 180,E1 -13140,E2 -13140} C_VEL
LIN {X 0,Y 362.284,Z 503.359,A -85,B 0,C 180,E1 -13142.224,E2 -13142.224} C_VEL
LIN {X 0,Y 362.129,Z 503.374,A -85,B 0,C 180,E1 -13146.687,E2 -13146.687} C_VEL
LIN {X 0,Y 362.035,Z 503.391,A -85,B 0,C 180,E1 -13150.062,E2 -13150.062} C_VEL
LIN {X 0,Y 362.023,Z 503.494,A -85,B 0,C 180,E1 -13154.128,E2 -13154.128} C_VEL
LIN {X 0,Y 365.534,Z 513.042,A -85,B 0,C 180,E1 -13155.044,E2 -13155.044} C_VEL
LIN {X 0,Y 368.897,Z 523.49,A -85,B 0,C 180,E1 -13156.179,E2 -13156.179} C_VEL
LIN {X 0,Y 369.522,Z 527.023,A -85,B 0,C 180,E1 -13156.576,E2 -13156.576} C_VEL
LIN {X 0,Y 368.55,Z 538.063,A -85,B 0,C 180,E1 -13157.765,E2 -13157.765} C_VEL
LIN {X 0,Y 367.573,Z 547.084,A -85,B 0,C 180,E1 -13158.968,E2 -13158.968} C_VEL
LIN {X 0,Y 366.465,Z 556.335,A -85,B 0,C 180,E1 -13160.487,E2 -13160.487} C_VEL
LIN {X 0,Y 365.524,Z 563.611,A -85,B 0,C 180,E1 -13161.961,E2 -13161.961} C_VEL
LIN {X 0,Y 364.618,Z 570.099,A -85,B 0,C 180,E1 -13163.576,E2 -13163.576} C_VEL
LIN {X 0,Y 363.921,Z 575.113,A -85,B 0,C 180,E1 -13165.142,E2 -13165.142} C_VEL
LIN {X 0,Y 363.173,Z 579.904,A -85,B 0,C 180,E1 -13167.104,E2 -13167.104} C_VEL
LIN {X 0,Y 362.609,Z 583.157,A -85,B 0,C 180,E1 -13168.983,E2 -13168.983} C_VEL
LIN {X 0,Y 362.342,Z 584.7,A -85,B 0,C 180,E1 -13170.285,E2 -13170.285} C_VEL
LIN {X 0,Y 362.126,Z 585.666,A -85,B 0,C 180,E1 -13171.602,E2 -13171.602} C_VEL
LIN {X 0,Y 361.94,Z 586.11,A -85,B 0,C 180,E1 -13173.388,E2 -13173.388} C_VEL
LIN {X 0,Y 361.897,Z 585.232,A -85,B 0,C 180,E1 -13175.634,E2 -13175.634} C_VEL
LIN {X 0,Y 361.955,Z 583.618,A -85,B 0,C 180,E1 -13177.241,E2 -13177.241} C_VEL
LIN {X 0,Y 362.172,Z 580.678,A -85,B 0,C 180,E1 -13179.085,E2 -13179.085} C_VEL
LIN {X 0,Y 362.673,Z 575.743,A -85,B 0,C 180,E1 -13181.214,E2 -13181.214} C_VEL
LIN {X 0,Y 363.173,Z 570.184,A -85,B 0,C 180,E1 -13183.012,E2 -13183.012} C_VEL
LIN {X 0,Y 363.866,Z 562.636,A -85,B 0,C 180,E1 -13184.902,E2 -13184.902} C_VEL
LIN {X 0,Y 364.647,Z 554.76,A -85,B 0,C 180,E1 -13186.479,E2 -13186.479} C_VEL
LIN {X 0,Y 365.345,Z 546.891,A -85,B 0,C 180,E1 -13187.781,E2 -13187.781} C_VEL
LIN {X 0,Y 366.178,Z 536.907,A -85,B 0,C 180,E1 -13189.142,E2 -13189.142} C_VEL
LIN {X 0,Y 366.909,Z 526.468,A -85,B 0,C 180,E1 -13190.292,E2 -13190.292} C_VEL
LIN {X 0,Y 367.17,Z 522.78,A -85,B 0,C 180,E1 -13190.646,E2 -13190.646} C_VEL
LIN {X 0,Y 364.784,Z 513.301,A -85,B 0,C 180,E1 -13191.587,E2 -13191.587} C_VEL
LIN {X 0,Y 361.872,Z 503.411,A -85,B 0,C 180,E1 -13192.431,E2 -13192.431} C_VEL
LIN {X 0,Y 361.859,Z 503.411,A -85,B 0,C 180,E1 -13195.72,E2 -13195.72} C_VEL
LIN {X 0,Y 361.88,Z 503.409,A -85,B 0,C 180,E1 -13199.672,E2 -13199.672} C_VEL
LIN {X 0,Y 361.959,Z 503.4,A -85,B 0,C 180,E1 -13203.475,E2 -13203.475} C_VEL
LIN {X 0,Y 361.884,Z 503.408,A -85,B 0,C 180,E1 -13207.144,E2 -13207.144} C_VEL
LIN {X 0,Y 361.891,Z 503.405,A -85,B 0,C 180,E1 -13210.722,E2 -13210.722} C_VEL
LIN {X 0,Y 361.949,Z 503.397,A -85,B 0,C 180,E1 -13214.226,E2 -13214.226} C_VEL
LIN {X 0,Y 362.004,Z 503.39,A -85,B 0,C 180,E1 -13216.528,E2 -13216.528} C_VEL
LIN {X 0,Y 362.005,Z 503.39,A -85,B 0,C 180,E1 -13219.937,E2 -13219.937} C_VEL
LIN {X 0,Y 362.129,Z 503.379,A -85,B 0,C 180,E1 -13223.313,E2 -13223.313} C_VEL
LIN {X 0,Y 362.285,Z 503.357,A -85,B 0,C 180,E1 -13227.776,E2 -13227.776} C_VEL
LIN {X 0,Y 362.365,Z 503.345,A -85,B 0,C 180,E1 -13230,E2 -13230} C_VEL
LIN {X 0,Y 362.283,Z 503.355,A -85,B 0,C 180,E1 -13232.223,E2 -13232.223} C_VEL
LIN {X 0,Y 362.129,Z 503.375,A -85,B 0,C 180,E1 -13236.687,E2 -13236.687} C_VEL
LIN {X 0,Y 362.005,Z 503.39,A -85,B 0,C 180,E1 -13240.063,E2 -13240.063} C_VEL
LIN {X 0,Y 362.003,Z 503.39,A -85,B 0,C 180,E1 -13243.899,E2 -13243.899} C_VEL
LIN {X 0,Y 361.933,Z 503.402,A -85,B 0,C 180,E1 -13246.934,E2 -13246.934} C_VEL
LIN {X 0,Y 361.898,Z 503.403,A -85,B 0,C 180,E1 -13250.46,E2 -13250.46} C_VEL
LIN {X 0,Y 361.897,Z 503.403,A -85,B 0,C 180,E1 -13254.112,E2 -13254.112} C_VEL
LIN {X 0,Y 361.868,Z 503.408,A -85,B 0,C 180,E1 -13257.782,E2 -13257.782} C_VEL
LIN {X 0,Y 361.851,Z 503.413,A -85,B 0,C 180,E1 -13261.285,E2 -13261.285} C_VEL
LIN {X 0,Y 361.858,Z 503.408,A -85,B 0,C 180,E1 -13264.28,E2 -13264.28} C_VEL
LIN {X 0,Y 361.864,Z 503.412,A -85,B 0,C 180,E1 -13267.222,E2 -13267.222} C_VEL
LIN {X 0,Y 361.815,Z 503.416,A -85,B 0,C 180,E1 -13270.751,E2 -13270.751} C_VEL
LIN {X 0,Y 361.827,Z 503.414,A -85,B 0,C 180,E1 -13272.95,E2 -13272.95} C_VEL
LIN {X 0,Y 361.132,Z 503.499,A -85,B 0,C 180,E1 -13273.879,E2 -13273.879} C_VEL
LIN {X 0,Y 358.301,Z 503.854,A -85,B 0,C 180,E1 -13275.391,E2 -13275.391} C_VEL
LIN {X 0,Y 355.914,Z 504.152,A -85,B 0,C 180,E1 -13276.614,E2 -13276.614} C_VEL
LIN {X 0,Y 354.877,Z 504.28,A -85,B 0,C 180,E1 -13277.56,E2 -13277.56} C_VEL
LIN {X 0,Y 354.784,Z 504.289,A -85,B 0,C 180,E1 -13277.88,E2 -13277.88} C_VEL
LIN {X 0,Y 354.818,Z 504.287,A -85,B 0,C 180,E1 -13280.666,E2 -13280.666} C_VEL
LIN {X 0,Y 354.824,Z 504.284,A -85,B 0,C 180,E1 -13284.3,E2 -13284.3} C_VEL
LIN {X 0,Y 354.79,Z 504.289,A -85,B 0,C 180,E1 -13287.666,E2 -13287.666} C_VEL
LIN {X 0,Y 354.871,Z 504.28,A -85,B 0,C 180,E1 -13290.621,E2 -13290.621} C_VEL
LIN {X 0,Y 354.9,Z 504.275,A -85,B 0,C 180,E1 -13294.172,E2 -13294.172} C_VEL
LIN {X 0,Y 354.818,Z 504.284,A -85,B 0,C 180,E1 -13297.892,E2 -13297.892} C_VEL
LIN {X 0,Y 354.925,Z 504.272,A -85,B 0,C 180,E1 -13301.891,E2 -13301.891} C_VEL
LIN {X 0,Y 354.945,Z 504.269,A -85,B 0,C 180,E1 -13305.981,E2 -13305.981} C_VEL
LIN {X 0,Y 354.959,Z 504.267,A -85,B 0,C 180,E1 -13309.735,E2 -13309.735} C_VEL
LIN {X 0,Y 355.102,Z 504.253,A -85,B 0,C 180,E1 -13313.18,E2 -13313.18} C_VEL
LIN {X 0,Y 355.243,Z 504.232,A -85,B 0,C 180,E1 -13317.732,E2 -13317.732} C_VEL
LIN {X 0,Y 355.354,Z 504.218,A -85,B 0,C 180,E1 -13320,E2 -13320} C_VEL
LIN {X 0,Y 355.234,Z 504.233,A -85,B 0,C 180,E1 -13322.267,E2 -13322.267} C_VEL
LIN {X 0,Y 355.091,Z 504.255,A -85,B 0,C 180,E1 -13326.82,E2 -13326.82} C_VEL
LIN {X 0,Y 354.982,Z 504.265,A -85,B 0,C 180,E1 -13330.264,E2 -13330.264} C_VEL
LIN {X 0,Y 354.945,Z 504.269,A -85,B 0,C 180,E1 -13334.019,E2 -13334.019} C_VEL
LIN {X 0,Y 354.891,Z 504.276,A -85,B 0,C 180,E1 -13338.092,E2 -13338.092} C_VEL
LIN {X 0,Y 354.818,Z 504.285,A -85,B 0,C 180,E1 -13342.107,E2 -13342.107} C_VEL
LIN {X 0,Y 354.828,Z 504.283,A -85,B 0,C 180,E1 -13345.833,E2 -13345.833} C_VEL
LIN {X 0,Y 354.8,Z 504.287,A -85,B 0,C 180,E1 -13349.683,E2 -13349.683} C_VEL
LIN {X 0,Y 354.787,Z 504.29,A -85,B 0,C 180,E1 -13352.333,E2 -13352.333} C_VEL
LIN {X 0,Y 354.822,Z 504.284,A -85,B 0,C 180,E1 -13355.699,E2 -13355.699} C_VEL
LIN {X 0,Y 354.825,Z 504.287,A -85,B 0,C 180,E1 -13359.423,E2 -13359.423} C_VEL
LIN {X 0,Y 354.804,Z 504.288,A -85,B 0,C 180,E1 -13363.33,E2 -13363.33} C_VEL
LIN {X 0,Y 354.825,Z 504.403,A -85,B 0,C 180,E1 -13363.817,E2 -13363.817} C_VEL
LIN {X 0,Y 356.603,Z 513.245,A -85,B 0,C 180,E1 -13367.408,E2 -13367.408} C_VEL
LIN {X 0,Y 358.475,Z 522.99,A -85,B 0,C 180,E1 -13371.144,E2 -13371.144} C_VEL
LIN {X 0,Y 358.983,Z 527.083,A -85,B 0,C 180,E1 -13372.634,E2 -13372.634} C_VEL
LIN {X 0,Y 357.792,Z 537.197,A -85,B 0,C 180,E1 -13376.08,E2 -13376.08} C_VEL
LIN {X 0,Y 356.826,Z 546.571,A -85,B 0,C 180,E1 -13379.197,E2 -13379.197} C_VEL
LIN {X 0,Y 355.764,Z 558.146,A -85,B 0,C 180,E1 -13382.976,E2 -13382.976} C_VEL
LIN {X 0,Y 354.955,Z 569.591,A -85,B 0,C 180,E1 -13386.672,E2 -13386.672} C_VEL
LIN {X 0,Y 354.409,Z 580.177,A -85,B 0,C 180,E1 -13390.035,E2 -13390.035} C_VEL
LIN {X 0,Y 355.989,Z 595.79,A -85,B 0,C 180,E1 -13390.687,E2 -13390.687} C_VEL
LIN {X 0,Y 356.824,Z 607.918,A -85,B 0,C 180,E1 -13391.393,E2 -13391.393} C_VEL
LIN {X 0,Y 357.407,Z 619.414,A -85,B 0,C 180,E1 -13392.255,E2 -13392.255} C_VEL
LIN {X 0,Y 357.571,Z 630.63,A -85,B 0,C 180,E1 -13393.295,E2 -13393.295} C_VEL
LIN {X 0,Y 356.533,Z 640.736,A -85,B 0,C 180,E1 -13394.42,E2 -13394.42} C_VEL
LIN {X 0,Y 355.597,Z 649.873,A -85,B 0,C 180,E1 -13395.664,E2 -13395.664} C_VEL
LIN {X 0,Y 354.888,Z 658.699,A -85,B 0,C 180,E1 -13397.127,E2 -13397.127} C_VEL
LIN {X 0,Y 354.305,Z 667.085,A -85,B 0,C 180,E1 -13398.849,E2 -13398.849} C_VEL
LIN {X 0,Y 354.035,Z 673.856,A -85,B 0,C 180,E1 -13400.574,E2 -13400.574} C_VEL
LIN {X 0,Y 353.953,Z 680.031,A -85,B 0,C 180,E1 -13402.585,E2 -13402.585} C_VEL
LIN {X 0,Y 354.036,Z 684.002,A -85,B 0,C 180,E1 -13404.304,E2 -13404.304} C_VEL
LIN {X 0,Y 354.255,Z 686.04,A -85,B 0,C 180,E1 -13405.449,E2 -13405.449} C_VEL
LIN {X 0,Y 354.285,Z 687.603,A -85,B 0,C 180,E1 -13406.588,E2 -13406.588} C_VEL
LIN {X 0,Y 354.333,Z 688.734,A -85,B 0,C 180,E1 -13407.727,E2 -13407.727} C_VEL
LIN {X 0,Y 354.646,Z 689.664,A -85,B 0,C 180,E1 -13410,E2 -13410} C_VEL
LIN {X 0,Y 354.313,Z 688.826,A -85,B 0,C 180,E1 -13412.274,E2 -13412.274} C_VEL
LIN {X 0,Y 354.253,Z 687.752,A -85,B 0,C 180,E1 -13413.412,E2 -13413.412} C_VEL
LIN {X 0,Y 354.177,Z 686.246,A -85,B 0,C 180,E1 -13414.553,E2 -13414.553} C_VEL
LIN {X 0,Y 353.969,Z 682.557,A -85,B 0,C 180,E1 -13416.544,E2 -13416.544} C_VEL
LIN {X 0,Y 353.912,Z 677.362,A -85,B 0,C 180,E1 -13418.565,E2 -13418.565} C_VEL
LIN {X 0,Y 354.11,Z 670.558,A -85,B 0,C 180,E1 -13420.579,E2 -13420.579} C_VEL
LIN {X 0,Y 354.652,Z 663.281,A -85,B 0,C 180,E1 -13422.3,E2 -13422.3} C_VEL
LIN {X 0,Y 355.363,Z 654.816,A -85,B 0,C 180,E1 -13423.938,E2 -13423.938} C_VEL
LIN {X 0,Y 356.465,Z 645.288,A -85,B 0,C 180,E1 -13425.436,E2 -13425.436} C_VEL
LIN {X 0,Y 357.607,Z 635.494,A -85,B 0,C 180,E1 -13426.704,E2 -13426.704} C_VEL
LIN {X 0,Y 358.226,Z 627.831,A -85,B 0,C 180,E1 -13427.556,E2 -13427.556} C_VEL
LIN {X 0,Y 358.338,Z 614.641,A -85,B 0,C 180,E1 -13428.801,E2 -13428.801} C_VEL
LIN {X 0,Y 358.032,Z 601.536,A -85,B 0,C 180,E1 -13429.792,E2 -13429.792} C_VEL
LIN {X 0,Y 356.788,Z 587.955,A -85,B 0,C 180,E1 -13430.616,E2 -13430.616} C_VEL
LIN {X 0,Y 354.472,Z 573.651,A -85,B 0,C 180,E1 -13431.346,E2 -13431.346} C_VEL
LIN {X 0,Y 355.131,Z 561.43,A -85,B 0,C 180,E1 -13435.181,E2 -13435.181} C_VEL
LIN {X 0,Y 355.973,Z 549.837,A -85,B 0,C 180,E1 -13438.928,E2 -13438.928} C_VEL
LIN {X 0,Y 357.04,Z 538.396,A -85,B 0,C 180,E1 -13442.773,E2 -13442.773} C_VEL
LIN {X 0,Y 358.333,Z 527.898,A -85,B 0,C 180,E1 -13446.473,E2 -13446.473} C_VEL
LIN {X 0,Y 358.577,Z 524.163,A -85,B 0,C 180,E1 -13447.87,E2 -13447.87} C_VEL
LIN {X 0,Y 357.394,Z 516.61,A -85,B 0,C 180,E1 -13451.008,E2 -13451.008} C_VEL
LIN {X 0,Y 355.78,Z 508.725,A -85,B 0,C 180,E1 -13454.673,E2 -13454.673} C_VEL
LIN {X 0,Y 354.792,Z 504.296,A -85,B 0,C 180,E1 -13457.016,E2 -13457.016} C_VEL
LIN {X 0,Y 354.817,Z 504.29,A -85,B 0,C 180,E1 -13460.666,E2 -13460.666} C_VEL
LIN {X 0,Y 354.824,Z 504.287,A -85,B 0,C 180,E1 -13464.301,E2 -13464.301} C_VEL
LIN {X 0,Y 354.789,Z 504.289,A -85,B 0,C 180,E1 -13467.667,E2 -13467.667} C_VEL
LIN {X 0,Y 354.871,Z 504.275,A -85,B 0,C 180,E1 -13470.622,E2 -13470.622} C_VEL
LIN {X 0,Y 354.902,Z 504.275,A -85,B 0,C 180,E1 -13474.173,E2 -13474.173} C_VEL
LIN {X 0,Y 354.838,Z 504.284,A -85,B 0,C 180,E1 -13477.894,E2 -13477.894} C_VEL
LIN {X 0,Y 354.925,Z 504.27,A -85,B 0,C 180,E1 -13481.892,E2 -13481.892} C_VEL
LIN {X 0,Y 354.946,Z 504.268,A -85,B 0,C 180,E1 -13485.981,E2 -13485.981} C_VEL
LIN {X 0,Y 354.981,Z 504.267,A -85,B 0,C 180,E1 -13489.736,E2 -13489.736} C_VEL
LIN {X 0,Y 355.118,Z 504.244,A -85,B 0,C 180,E1 -13492.037,E2 -13492.037} C_VEL
LIN {X 0,Y 355.094,Z 504.253,A -85,B 0,C 180,E1 -13494.321,E2 -13494.321} C_VEL
LIN {X 0,Y 355.237,Z 504.234,A -85,B 0,C 180,E1 -13497.733,E2 -13497.733} C_VEL
LIN {X 0,Y 355.377,Z 504.218,A -85,B 0,C 180,E1 -13500,E2 -13500} C_VEL
LIN {X 0,Y 355.247,Z 504.235,A -85,B 0,C 180,E1 -13502.268,E2 -13502.268} C_VEL
LIN {X 0,Y 355.094,Z 504.251,A -85,B 0,C 180,E1 -13506.82,E2 -13506.82} C_VEL
LIN {X 0,Y 354.982,Z 504.269,A -85,B 0,C 180,E1 -13510.264,E2 -13510.264} C_VEL
LIN {X 0,Y 354.99,Z 504.435,A -85,B 0,C 180,E1 -13513.598,E2 -13513.598} C_VEL
LIN {X 0,Y 356.978,Z 509.719,A -85,B 0,C 180,E1 -13514.103,E2 -13514.103} C_VEL
LIN {X 0,Y 360.817,Z 520.273,A -85,B 0,C 180,E1 -13515.246,E2 -13515.246} C_VEL
LIN {X 0,Y 362.913,Z 528.165,A -85,B 0,C 180,E1 -13516.178,E2 -13516.178} C_VEL
LIN {X 0,Y 362.008,Z 538.738,A -85,B 0,C 180,E1 -13517.335,E2 -13517.335} C_VEL
LIN {X 0,Y 360.813,Z 549.077,A -85,B 0,C 180,E1 -13518.748,E2 -13518.748} C_VEL
LIN {X 0,Y 359.677,Z 558.179,A -85,B 0,C 180,E1 -13520.296,E2 -13520.296} C_VEL
LIN {X 0,Y 358.653,Z 565.576,A -85,B 0,C 180,E1 -13521.859,E2 -13521.859} C_VEL
LIN {X 0,Y 357.574,Z 572.699,A -85,B 0,C 180,E1 -13523.761,E2 -13523.761} C_VEL
LIN {X 0,Y 356.663,Z 578.273,A -85,B 0,C 180,E1 -13525.691,E2 -13525.691} C_VEL
LIN {X 0,Y 356.125,Z 581.892,A -85,B 0,C 180,E1 -13527.369,E2 -13527.369} C_VEL
LIN {X 0,Y 355.833,Z 583.475,A -85,B 0,C 180,E1 -13528.296,E2 -13528.296} C_VEL
LIN {X 0,Y 355.472,Z 585.208,A -85,B 0,C 180,E1 -13529.622,E2 -13529.622} C_VEL
LIN {X 0,Y 355.103,Z 586.825,A -85,B 0,C 180,E1 -13531.675,E2 -13531.675} C_VEL
LIN {X 0,Y 354.904,Z 587.137,A -85,B 0,C 180,E1 -13533.725,E2 -13533.725} C_VEL
LIN {X 0,Y 354.869,Z 586.187,A -85,B 0,C 180,E1 -13535.709,E2 -13535.709} C_VEL
LIN {X 0,Y 354.98,Z 583.791,A -85,B 0,C 180,E1 -13537.862,E2 -13537.862} C_VEL
LIN {X 0,Y 355.342,Z 579.771,A -85,B 0,C 180,E1 -13540.059,E2 -13540.059} C_VEL
LIN {X 0,Y 355.885,Z 574.228,A -85,B 0,C 180,E1 -13542.178,E2 -13542.178} C_VEL
LIN {X 0,Y 356.488,Z 568.198,A -85,B 0,C 180,E1 -13543.944,E2 -13543.944} C_VEL
LIN {X 0,Y 357.135,Z 561.549,A -85,B 0,C 180,E1 -13545.51,E2 -13545.51} C_VEL
LIN {X 0,Y 358.024,Z 552.687,A -85,B 0,C 180,E1 -13547.196,E2 -13547.196} C_VEL
LIN {X 0,Y 358.844,Z 542.788,A -85,B 0,C 180,E1 -13548.727,E2 -13548.727} C_VEL
LIN {X 0,Y 359.707,Z 531.959,A -85,B 0,C 180,E1 -13550.063,E2 -13550.063} C_VEL
LIN {X 0,Y 360.289,Z 524.442,A -85,B 0,C 180,E1 -13550.837,E2 -13550.837} C_VEL
LIN {X 0,Y 359.087,Z 519.04,A -85,B 0,C 180,E1 -13551.402,E2 -13551.402} C_VEL
LIN {X 0,Y 355.872,Z 507.956,A -85,B 0,C 180,E1 -13552.436,E2 -13552.436} C_VEL
LIN {X 0,Y 354.846,Z 504.286,A -85,B 0,C 180,E1 -13552.759,E2 -13552.759} C_VEL
LIN {X 0,Y 354.819,Z 504.285,A -85,B 0,C 180,E1 -13556.316,E2 -13556.316} C_VEL
LIN {X 0,Y 354.859,Z 504.28,A -85,B 0,C 180,E1 -13560.322,E2 -13560.322} C_VEL
LIN {X 0,Y 354.903,Z 504.275,A -85,B 0,C 180,E1 -13564.173,E2 -13564.173} C_VEL
LIN {X 0,Y 354.821,Z 504.286,A -85,B 0,C 180,E1 -13567.893,E2 -13567.893} C_VEL
LIN {X 0,Y 354.895,Z 504.276,A -85,B 0,C 180,E1 -13571.908,E2 -13571.908} C_VEL
LIN {X 0,Y 354.948,Z 504.27,A -85,B 0,C 180,E1 -13575.981,E2 -13575.981} C_VEL
LIN {X 0,Y 354.961,Z 504.269,A -85,B 0,C 180,E1 -13579.735,E2 -13579.735} C_VEL
LIN {X 0,Y 355.094,Z 504.255,A -85,B 0,C 180,E1 -13583.18,E2 -13583.18} C_VEL
LIN {X 0,Y 355.249,Z 504.233,A -85,B 0,C 180,E1 -13587.732,E2 -13587.732} C_VEL
LIN {X 0,Y 355.316,Z 504.223,A -85,B 0,C 180,E1 -13590,E2 -13590} C_VEL
LIN {X 0,Y 355.246,Z 504.231,A -85,B 0,C 180,E1 -13592.267,E2 -13592.267} C_VEL
LIN {X 0,Y 355.094,Z 504.252,A -85,B 0,C 180,E1 -13596.82,E2 -13596.82} C_VEL
LIN {X 0,Y 354.961,Z 504.267,A -85,B 0,C 180,E1 -13600.264,E2 -13600.264} C_VEL
LIN {X 0,Y 354.948,Z 504.269,A -85,B 0,C 180,E1 -13604.019,E2 -13604.019} C_VEL
LIN {X 0,Y 354.894,Z 504.275,A -85,B 0,C 180,E1 -13608.092,E2 -13608.092} C_VEL
LIN {X 0,Y 354.837,Z 504.283,A -85,B 0,C 180,E1 -13612.106,E2 -13612.106} C_VEL
LIN {X 0,Y 354.868,Z 504.279,A -85,B 0,C 180,E1 -13615.83,E2 -13615.83} C_VEL
LIN {X 0,Y 354.811,Z 504.287,A -85,B 0,C 180,E1 -13619.682,E2 -13619.682} C_VEL
LIN {X 0,Y 354.818,Z 504.286,A -85,B 0,C 180,E1 -13623.684,E2 -13623.684} C_VEL
LIN {X 0,Y 354.799,Z 504.288,A -85,B 0,C 180,E1 -13626.459,E2 -13626.459} C_VEL
LIN {X 0,Y 354.771,Z 504.294,A -85,B 0,C 180,E1 -13629.412,E2 -13629.412} C_VEL
LIN {X 0,Y 354.783,Z 504.292,A -85,B 0,C 180,E1 -13632.938,E2 -13632.938} C_VEL
LIN {X 0,Y 354.769,Z 504.291,A -85,B 0,C 180,E1 -13636.103,E2 -13636.103} C_VEL
LIN {X 0,Y 354.784,Z 504.289,A -85,B 0,C 180,E1 -13637.88,E2 -13637.88} C_VEL
LIN {X 0,Y 354.101,Z 504.378,A -85,B 0,C 180,E1 -13638.828,E2 -13638.828} C_VEL
LIN {X 0,Y 351.27,Z 504.731,A -85,B 0,C 180,E1 -13640.37,E2 -13640.37} C_VEL
LIN {X 0,Y 348.878,Z 505.03,A -85,B 0,C 180,E1 -13641.618,E2 -13641.618} C_VEL
LIN {X 0,Y 347.843,Z 505.156,A -85,B 0,C 180,E1 -13642.584,E2 -13642.584} C_VEL
LIN {X 0,Y 347.752,Z 505.165,A -85,B 0,C 180,E1 -13642.91,E2 -13642.91} C_VEL
LIN {X 0,Y 347.751,Z 505.165,A -85,B 0,C 180,E1 -13645.956,E2 -13645.956} C_VEL
LIN {X 0,Y 347.767,Z 505.164,A -85,B 0,C 180,E1 -13649.653,E2 -13649.653} C_VEL
LIN {X 0,Y 347.853,Z 505.155,A -85,B 0,C 180,E1 -13652.745,E2 -13652.745} C_VEL
LIN {X 0,Y 347.787,Z 505.16,A -85,B 0,C 180,E1 -13656.161,E2 -13656.161} C_VEL
LIN {X 0,Y 347.809,Z 505.158,A -85,B 0,C 180,E1 -13659.909,E2 -13659.909} C_VEL
LIN {X 0,Y 347.869,Z 505.151,A -85,B 0,C 180,E1 -13662.359,E2 -13662.359} C_VEL
LIN {X 0,Y 347.9,Z 505.146,A -85,B 0,C 180,E1 -13665.97,E2 -13665.97} C_VEL
LIN {X 0,Y 347.899,Z 505.147,A -85,B 0,C 180,E1 -13669.524,E2 -13669.524} C_VEL
LIN {X 0,Y 348.07,Z 505.13,A -85,B 0,C 180,E1 -13673.041,E2 -13673.041} C_VEL
LIN {X 0,Y 348.205,Z 505.109,A -85,B 0,C 180,E1 -13677.686,E2 -13677.686} C_VEL
LIN {X 0,Y 348.305,Z 505.096,A -85,B 0,C 180,E1 -13680,E2 -13680} C_VEL
LIN {X 0,Y 348.196,Z 505.11,A -85,B 0,C 180,E1 -13682.313,E2 -13682.313} C_VEL
LIN {X 0,Y 348.058,Z 505.132,A -85,B 0,C 180,E1 -13686.958,E2 -13686.958} C_VEL
LIN {X 0,Y 347.933,Z 505.145,A -85,B 0,C 180,E1 -13690.474,E2 -13690.474} C_VEL
LIN {X 0,Y 347.9,Z 505.147,A -85,B 0,C 180,E1 -13694.15,E2 -13694.15} C_VEL
LIN {X 0,Y 347.83,Z 505.156,A -85,B 0,C 180,E1 -13698.259,E2 -13698.259} C_VEL
LIN {X 0,Y 347.77,Z 505.163,A -85,B 0,C 180,E1 -13701.626,E2 -13701.626} C_VEL
LIN {X 0,Y 347.777,Z 505.165,A -85,B 0,C 180,E1 -13705.111,E2 -13705.111} C_VEL
LIN {X 0,Y 347.741,Z 505.166,A -85,B 0,C 180,E1 -13707.7,E2 -13707.7} C_VEL
LIN {X 0,Y 347.741,Z 505.168,A -85,B 0,C 180,E1 -13710.349,E2 -13710.349} C_VEL
LIN {X 0,Y 347.749,Z 505.166,A -85,B 0,C 180,E1 -13714.044,E2 -13714.044} C_VEL
LIN {X 0,Y 347.762,Z 505.164,A -85,B 0,C 180,E1 -13717.321,E2 -13717.321} C_VEL
LIN {X 0,Y 347.733,Z 505.171,A -85,B 0,C 180,E1 -13720.297,E2 -13720.297} C_VEL
LIN {X 0,Y 347.78,Z 505.257,A -85,B 0,C 180,E1 -13723.449,E2 -13723.449} C_VEL
LIN {X 0,Y 349.67,Z 514.642,A -85,B 0,C 180,E1 -13727.34,E2 -13727.34} C_VEL
LIN {X 0,Y 351.569,Z 524.597,A -85,B 0,C 180,E1 -13731.226,E2 -13731.226} C_VEL
LIN {X 0,Y 352.002,Z 527.919,A -85,B 0,C 180,E1 -13732.467,E2 -13732.467} C_VEL
LIN {X 0,Y 350.8,Z 537.72,A -85,B 0,C 180,E1 -13735.878,E2 -13735.878} C_VEL
LIN {X 0,Y 349.761,Z 547.423,A -85,B 0,C 180,E1 -13739.177,E2 -13739.177} C_VEL
LIN {X 0,Y 348.668,Z 558.995,A -85,B 0,C 180,E1 -13743.051,E2 -13743.051} C_VEL
LIN {X 0,Y 347.838,Z 570.362,A -85,B 0,C 180,E1 -13746.797,E2 -13746.797} C_VEL
LIN {X 0,Y 347.364,Z 579.26,A -85,B 0,C 180,E1 -13749.689,E2 -13749.689} C_VEL
LIN {X 0,Y 348.946,Z 594.978,A -85,B 0,C 180,E1 -13750.363,E2 -13750.363} C_VEL
LIN {X 0,Y 349.83,Z 606.942,A -85,B 0,C 180,E1 -13751.077,E2 -13751.077} C_VEL
LIN {X 0,Y 350.414,Z 619.403,A -85,B 0,C 180,E1 -13752.039,E2 -13752.039} C_VEL
LIN {X 0,Y 350.567,Z 630.433,A -85,B 0,C 180,E1 -13753.101,E2 -13753.101} C_VEL
LIN {X 0,Y 349.448,Z 641.53,A -85,B 0,C 180,E1 -13754.396,E2 -13754.396} C_VEL
LIN {X 0,Y 348.411,Z 650.443,A -85,B 0,C 180,E1 -13755.68,E2 -13755.68} C_VEL
LIN {X 0,Y 347.761,Z 658.872,A -85,B 0,C 180,E1 -13757.156,E2 -13757.156} C_VEL
LIN {X 0,Y 347.198,Z 667.055,A -85,B 0,C 180,E1 -13758.913,E2 -13758.913} C_VEL
LIN {X 0,Y 346.943,Z 673.645,A -85,B 0,C 180,E1 -13760.674,E2 -13760.674} C_VEL
LIN {X 0,Y 346.884,Z 678.859,A -85,B 0,C 180,E1 -13762.433,E2 -13762.433} C_VEL
LIN {X 0,Y 346.97,Z 682.87,A -85,B 0,C 180,E1 -13764.187,E2 -13764.187} C_VEL
LIN {X 0,Y 347.184,Z 684.924,A -85,B 0,C 180,E1 -13765.356,E2 -13765.356} C_VEL
LIN {X 0,Y 347.244,Z 686.506,A -85,B 0,C 180,E1 -13766.519,E2 -13766.519} C_VEL
LIN {X 0,Y 347.299,Z 687.657,A -85,B 0,C 180,E1 -13767.681,E2 -13767.681} C_VEL
LIN {X 0,Y 347.378,Z 688.346,A -85,B 0,C 180,E1 -13768.841,E2 -13768.841} C_VEL
LIN {X 0,Y 347.619,Z 688.621,A -85,B 0,C 180,E1 -13770,E2 -13770} C_VEL
LIN {X 0,Y 347.271,Z 687.808,A -85,B 0,C 180,E1 -13772.32,E2 -13772.32} C_VEL
LIN {X 0,Y 347.205,Z 686.751,A -85,B 0,C 180,E1 -13773.482,E2 -13773.482} C_VEL
LIN {X 0,Y 347.111,Z 685.255,A -85,B 0,C 180,E1 -13774.646,E2 -13774.646} C_VEL
LIN {X 0,Y 346.866,Z 681.182,A -85,B 0,C 180,E1 -13776.874,E2 -13776.874} C_VEL
LIN {X 0,Y 346.838,Z 676.446,A -85,B 0,C 180,E1 -13778.741,E2 -13778.741} C_VEL
LIN {X 0,Y 347.05,Z 669.673,A -85,B 0,C 180,E1 -13780.797,E2 -13780.797} C_VEL
LIN {X 0,Y 347.63,Z 662.432,A -85,B 0,C 180,E1 -13782.553,E2 -13782.553} C_VEL
LIN {X 0,Y 348.308,Z 655.148,A -85,B 0,C 180,E1 -13784.013,E2 -13784.013} C_VEL
LIN {X 0,Y 349.34,Z 646.533,A -85,B 0,C 180,E1 -13785.46,E2 -13785.46} C_VEL
